// ---- GlobalTextList.TcGTLO
TEXTLIST GlobalTextList
  808 = '  +'
  159 = '  -'
  440 = ' +'
  1026 = ' -'
  1635 = '%0.2f'
  824 = '%i'
  778 = '+'
  2003 = '-'
  1760 = '1'
  225 = '2'
  751 = 'ACTUADORES'
  905 = 'Almacen'
  381 = 'Almacén'
  135 = 'Automático'
  67 = 'Azul'
  613 = 'Belt_Conveyor_2m_1'
  919 = 'Belt_conveyor_2m_1'
  114 = 'Belt_Conveyor_2m_2'
  119 = 'Belt_Conveyor_2m_3'
  170 = 'Belt_Conveyor_2m_4'
  987 = 'Belt_Conveyor_2m_5'
  96 = 'Belt_Conveyor_2m_6'
  269 = 'Belt_Conveyor_2m_7'
  285 = 'Belt_Conveyor_2m_8'
  759 = 'Belt_conveyor_4m_1'
  776 = 'Belt_Conveyor_4m_3'
  836 = 'Belt_Conveyor_4m_4'
  755 = 'Belt_Conveyor_4m_5'
  724 = 'Belt_Conveyor_4m_6'
  643 = 'Belt_conveyor_6m_1'
  497 = 'Belt_Conveyor_6m_2'
  202 = 'Belt_conveyor_6m_4'
  731 = 'Belt_conveyor_6m_5'
  768 = 'Belt_Conveyor_Inclined_1'
  535 = 'BL'
  1577 = 'Brazo'
  234 = 'Chain_Transfer_1_+'
  916 = 'Cinturon +'
  165 = 'Cinturón -'
  278 = 'Clamped base'
  1647 = 'Clamped der'
  321 = 'Clamped izq'
  82 = 'Clamped top'
  420 = 'Comienzo Linea Azul'
  1467 = 'Comienzo Produccion'
  78 = 'Comienzo Producción Azul'
  1309 = 'Command'
  1035 = 'Command ID'
  1959 = 'Control Almacen'
  1204 = 'Control Machines Centers'
  429 = 'Curved_Belt_Conveyor_1_CW'
  62 = 'Curved_Belt_Conveyor_2_CCW'
  578 = 'Curved_Roller_Conveyor_1_ccw'
  624 = 'Curved_Roller_Conveyor_2_ccw'
  222 = 'Descarte'
  1837 = 'Diffuse_Sensor_0'
  448 = 'Diffuse_Sensor_1'
  935 = 'Diffuse_Sensor_2'
  516 = 'Diffuse_Sensor_3'
  913 = 'Diffuse_Sensor_39'
  816 = 'Diffuse_Sensor_4'
  1082 = 'Diffuse_Sensor_41'
  895 = 'Diffuse_Sensor_43'
  528 = 'Diffuse_Sensor_44'
  482 = 'Diffuse_Sensor_5'
  68 = 'Diffuse_Sensor_8'
  560 = 'Emergency Stop'
  121 = 'Emergency Stop_1'
  284 = 'Emergency Stop_2'
  433 = 'Emisión'
  952 = 'Emisor'
  925 = 'Entrada'
  355 = 'Entrada Almacen'
  36 = 'Error RFID'
  683 = 'Extracción'
  1129 = 'f'
  120 = 'Final Linea Azul'
  1722 = 'Final Producción Azul'
  1140 = 'FL'
  296 = 'Flujo'
  363 = 'G'
  176 = 'gggg'
  131 = 'Giro Brazo'
  1627 = 'Giro Cinturon +'
  644 = 'Global'
  1976 = 'Grua'
  414 = 'hhhh'
  534 = 'inea Verde'
  546 = 'L'
  426 = 'Linea Almacen'
  588 = 'Linea Azul'
  456 = 'Linea Metal'
  439 = 'Linea Verde'
  1440 = 'Loading_Conveyor_1'
  1444 = 'Línea Almacén'
  386 = 'Machining_Center_1_Error'
  558 = 'Machining_Center_1_IsBusy'
  780 = 'Machining_Center_1_Opened'
  323 = 'Machining_Center_1_Produce_Lids'
  520 = 'Machining_Center_1_Progress'
  183 = 'Machining_Center_2_Error'
  615 = 'Machining_Center_2_IsBusy'
  617 = 'Machining_Center_2_Opened'
  1000 = 'Machining_Center_2_Produce_Lids'
  413 = 'Machining_Center_2_Progress'
  888 = 'Manual'
  1021 = 'Memory Index'
  1807 = 'ML'
  809 = 'Open_Door'
  105 = 'Open_Door_1'
  19 = 'Open_Door_2'
  976 = 'Palletizer'
  334 = 'Palletizer_1_Back_Limit'
  602 = 'Palletizer_1_Belt+'
  1173 = 'Palletizer_1_Belt-'
  536 = 'Palletizer_1_Chain+'
  942 = 'Palletizer_1_Chain-'
  1048 = 'Palletizer_1_Clamp'
  182 = 'Palletizer_1_Clamped'
  847 = 'Palletizer_1_Elevator+'
  108 = 'Palletizer_1_Elevator-'
  61 = 'Palletizer_1_Elevator_Moving'
  599 = 'Palletizer_1_Front_Limit'
  587 = 'Palletizer_1_MoveToLimit'
  124 = 'Palletizer_1_Open_Plate'
  557 = 'Palletizer_1_Plate_Limit'
  965 = 'Palletizer_1_Push'
  361 = 'Palletizer_1_Pusher_Limit'
  418 = 'Palletizer_1_Turn'
  404 = 'Pantalla Principal'
  897 = 'Pick & Place'
  1779 = 'Pinza'
  480 = 'Pivot_Arm_Sorter_1_Belt+'
  784 = 'Pivot_Arm_Sorter_1_Belt-'
  929 = 'Pivot_Arm_Sorter_1_Turn'
  302 = 'Pivot_Arm_Sorter_2_Belt+'
  744 = 'Pivot_Arm_Sorter_2_Belt-'
  614 = 'Pivot_Arm_Sorter_2_Turn'
  719 = 'Posición'
  762 = 'Principal'
  88 = 'Pusher_1'
  657 = 'Pusher_1_Back_Limit'
  45 = 'Pusher_1_Front_Limit'
  934 = 'Pusher_2'
  621 = 'Pusher_2_Back_Limit'
  774 = 'Pusher_2_Front_Limit'
  140 = 'Pusher_3'
  585 = 'Pusher_3_Back_Limit'
  306 = 'Pusher_3_Front_Limit'
  1770 = 'R'
  411 = 'Read Data'
  111 = 'Reset'
  1365 = 'Retroreflective_Sensor_1'
  331 = 'Retroreflective_Sensor_2'
  308 = 'RFID_Reader_1_Command'
  899 = 'RFID_Reader_1_Command_ID'
  459 = 'RFID_Reader_1_Ejecute_Command'
  1031 = 'RFID_Reader_1_Memory_Data'
  817 = 'RFID_Reader_1_Read_Data'
  377 = 'RFID_Reader_1_Status'
  874 = 'RFID_Reader_1_Writead_Data'
  508 = 'RFID_Reader_1_Write_Data'
  569 = 'Right_Positioner_1_Clamp'
  850 = 'Right_Positioner_1_Clamped'
  989 = 'Right_Positioner_1_Limit'
  523 = 'Right_Positioner_1_Raise'
  511 = 'Right_Positioner_2_Clamped'
  14 = 'Right_Positioner_2_Limit'
  620 = 'Roller_Conveyor_2m_1'
  251 = 'Roller_Conveyor_2m_2'
  1642 = 'Roller_Conveyor_2m_5'
  97 = 'Roller_Conveyor_2m_8'
  29 = 'Roller_Conveyor_4m_1'
  855 = 'Roller_Conveyor_4m_2'
  960 = 'Roller_Conveyor_4m_3'
  653 = 'Roller_Conveyor_6m_1'
  1263 = 'Roller_Conveyor_6m_2'
  627 = 'SENSORES'
  790 = 'Señales'
  1143 = 'Stacker_Crane_Left'
  1650 = 'Stacker_Crane_Left_Limit'
  1364 = 'Stacker_Crane_Lift'
  1622 = 'Stacker_Crane_Middle_Limit'
  1210 = 'Stacker_Crane_Moving_X'
  953 = 'Stacker_Crane_Moving_Z'
  1284 = 'Stacker_Crane_Right'
  380 = 'Stacker_Crane_Right_Limit'
  46 = 'Start'
  1155 = 'Start_1'
  1180 = 'Start_2'
  1706 = 'Status'
  769 = 'Stop'
  1228 = 'Stop_1'
  431 = 'Stop_2'
  518 = 'Turntable_1_Back_Limit'
  666 = 'Turntable_1_Front_Limit'
  556 = 'Turntable_1_Limit_0'
  77 = 'Turntable_1_Limit_90'
  1318 = 'Turntable_1_Roll_+'
  292 = 'Turntable_1_Roll_-'
  1288 = 'Turntable_1_Turn'
  1524 = 'Turntable_2_Back_Limit'
  1270 = 'Turntable_2_Front_Limit'
  235 = 'Turntable_2_Limit_0'
  473 = 'Turntable_2_Limit_90'
  1052 = 'Turntable_2_Roll_+'
  552 = 'Turntable_2_Roll_-'
  1580 = 'Turntable_2_Turn'
  337 = 'Two-Axis_Pick_Place_1_Detected'
  814 = 'Two-Axis_Pick_Place_1_Grab'
  112 = 'Two-Axis_Pick_Place_1_Gripper_CCW'
  309 = 'Two-Axis_Pick_Place_1_Gripper_CW'
  956 = 'Two-Axis_Pick_Place_1_Gripper_Rotating'
  811 = 'Two-Axis_Pick_Place_1_Moving_X'
  353 = 'Two-Axis_Pick_Place_1_Moving_Z'
  870 = 'Two-Axis_Pick_Place_1_Rotate'
  893 = 'Two-Axis_Pick_Place_1_Rotate_CCW'
  681 = 'Two-Axis_Pick_Place_1_Rotate_CW'
  541 = 'Two-Axis_Pick_Place_1_Rotating'
  568 = 'Two-Axis_Pick_Place_1_X'
  184 = 'Two-Axis_Pick_Place_1_Z'
  1262 = 'Two_Axis_Pick&Place'
  356 = 'Variables'
  810 = 'Vision_Sensor_1'
  288 = 'Vision_Sensor_10'
  21 = 'Vision_Sensor_11'
  936 = 'Vision_Sensor_12'
  53 = 'Vision_Sensor_13'
  669 = 'Vision_Sensor_14'
  985 = 'Vision_Sensor_15'
  999 = 'Vision_Sensor_4'
  357 = 'Vision_Sensor_40'
  996 = 'Vision_Sensor_42'
  84 = 'Vision_Sensor_5'
  841 = 'Vision_Sensor_6'
  335 = 'Vision_Sensor_7'
  688 = 'Vision_Sensor_8'
  43 = 'Vision_Sensor_9'
  1093 = 'vvvvvvvv'
  1646 = 'Write Data'
  1531 = 'Zona Inferior'
  909 = 'Zona Superior'
  805 = '¿Como introduzco valores?'
END_TEXTLIST

// ---- VISUs/Manual/Almacen_Manual.TcVIS
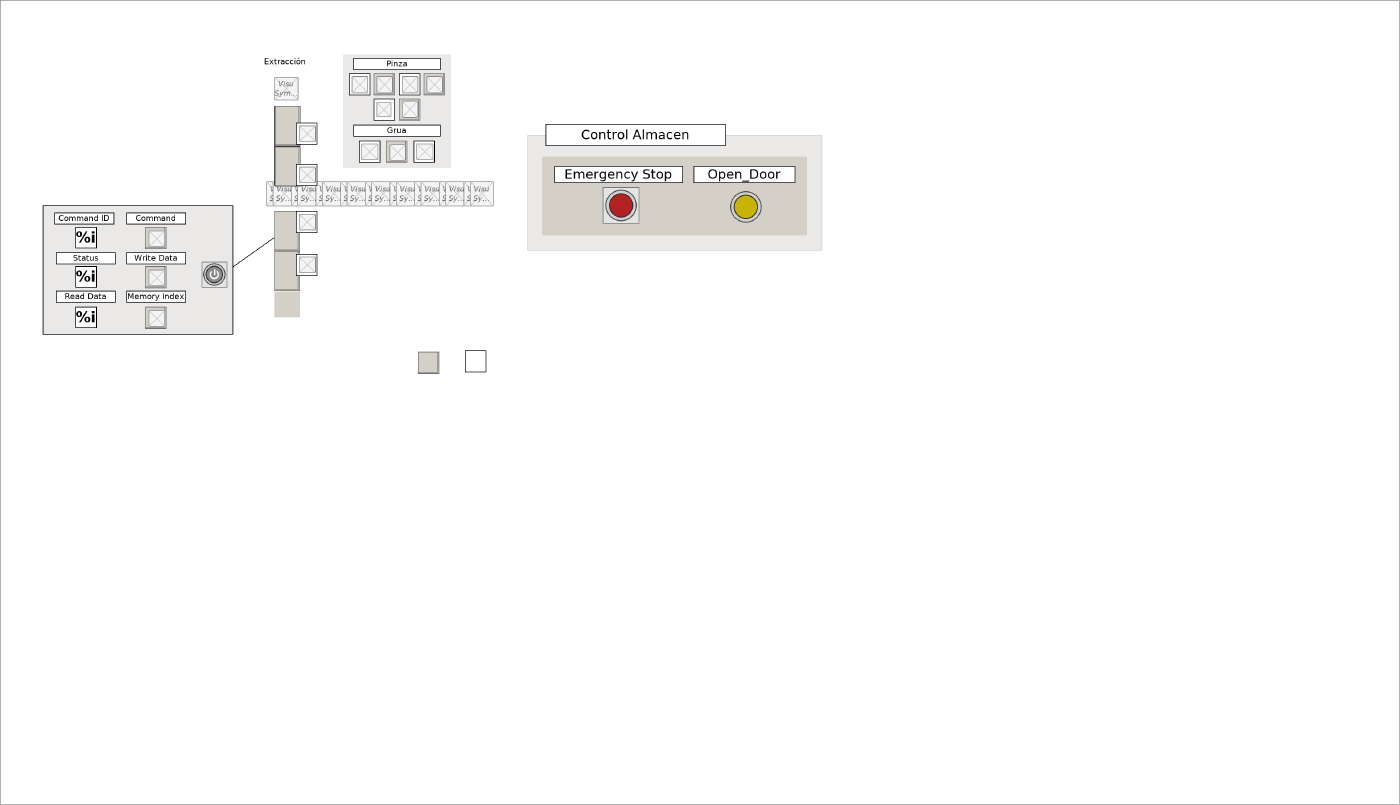
VISUALIZATION Almacen_Manual  // 1930x1110
    Rectangle (369,356 55x35), angle 90
    Group (367,250 330x48)
        Group (0,0 126x48)
            Group (0,0 92x48)
                Group (0,0 58x48)
                    Rectangle (8,5 24x23)
                    Image (0,0 32x34), image: VisuSymbols.Symbols.ArrowForward
                    Image (9,0 32x34), angle 90, image: VisuSymbols.Symbols.ArrowDown
                Group (34,0 58x48)
                    Rectangle (8,5 24x23)
                    Image (0,0 32x34), image: VisuSymbols.Symbols.ArrowForward
                    Image (9,0 32x34), angle 90, image: VisuSymbols.Symbols.ArrowDown
            Group (68,0 58x48)
                Rectangle (8,5 24x23)
                Image (0,0 32x34), image: VisuSymbols.Symbols.ArrowForward
                Image (9,0 32x34), angle 90, image: VisuSymbols.Symbols.ArrowDown
        Group (102,0 126x48)
            Group (0,0 92x48)
                Group (0,0 58x48)
                    Rectangle (8,5 24x23)
                    Image (0,0 32x34), image: VisuSymbols.Symbols.ArrowForward
                    Image (9,0 32x34), angle 90, image: VisuSymbols.Symbols.ArrowDown
                Group (34,0 58x48)
                    Rectangle (8,5 24x23)
                    Image (0,0 32x34), image: VisuSymbols.Symbols.ArrowForward
                    Image (9,0 32x34), angle 90, image: VisuSymbols.Symbols.ArrowDown
            Group (68,0 58x48)
                Rectangle (8,5 24x23)
                Image (0,0 32x34), image: VisuSymbols.Symbols.ArrowForward
                Image (9,0 32x34), angle 90, image: VisuSymbols.Symbols.ArrowDown
        Group (204,0 126x48)
            Group (0,0 92x48)
                Group (0,0 58x48)
                    Rectangle (8,5 24x23)
                    Image (0,0 32x34), image: VisuSymbols.Symbols.ArrowForward
                    Image (9,0 32x34), angle 90, image: VisuSymbols.Symbols.ArrowDown
                Group (34,0 58x48)
                    Rectangle (8,5 24x23)
                    Image (0,0 32x34), image: VisuSymbols.Symbols.ArrowForward
                    Image (9,0 32x34), angle 90, image: VisuSymbols.Symbols.ArrowDown
            Group (68,0 58x48)
                Rectangle (8,5 24x23)
                Image (0,0 32x34), image: VisuSymbols.Symbols.ArrowForward
                Image (9,0 32x34), angle 90, image: VisuSymbols.Symbols.ArrowDown
    InvisibleInput (355,103 77x35)
    Image (378,106 33x32), image: VisuSymbols.Symbols.ForwardStandard
    Rectangle (347,76 92x18), "Extracción"
    Rectangle (379,402 35x35), angle 90
    Rectangle (369,301 55x35), angle 90
    Rectangle (369,211 55x35), angle 90
    Rectangle (369,156 55x35), angle 90
    InvisibleInput (1163,198 18x136)
    Line (377,328) (318,370)
    InvisibleInput (262,497 18x41)
    Rectangle (1771,538 159x406), angle 90
    Rectangle (752,171 248x30), "Control Almacen"
    Rectangle (1780,528 108x365), angle 90
    PushSwitch (831,258 50x50), variable: GVL.Emergency_Stop_9, behaviour: TOGGLE, style: Switch-PushSwitch-Red
    Rectangle (764,229 177x23), "Emergency Stop"
    Lamp1 (1003,260 50x50), variable: NOT GVL.Safety_Door_13 OR NOT GVL.Safety_Door_14 OR NOT GVL.Safety_Door_15, style: Lamp-Lamp1-Yellow
    Rectangle (956,229 140x23), "Open_Door"
    Rectangle (1198,848 178x262), angle 90
    Rectangle (104,313 29x29), "%i", text variable: GVL.RFID_Reader_1_Command_ID
        p4168582468: GVL.RFID_Reader_1_Command_ID
    Rectangle (75,293 82x16), "Command ID"
    Rectangle (77,348 82x16), "Status"
    Rectangle (77,401 82x16), "Read Data"
    Rectangle (104,367 29x29), "%i", text variable: GVL.RFID_Reader_1_Status
        p4168582468: GVL.RFID_Reader_1_Status
    Rectangle (104,423 29x29), "%i", text variable: GVL.RFID_Reader_1_Read_Data
        p4168582468: GVL.RFID_Reader_1_Read_Data
    PowerSwitch (278,361 35x35), variable: GVL.RFID_Reader_1_Ejecute_Comm, behaviour: TOGGLE, style: Switch-PowerSwitch-Gray
    Button (378,346 35x55), colour toggle: GVL.Roller_Conveyor_2m_8, pressed state: GVL.Roller_Conveyor_2m_8
        OnMouseClick: toggle GVL.Roller_Conveyor_2m_8
    Button (378,291 35x55), colour toggle: GVL.Loading_Conveyor_1, pressed state: GVL.Loading_Conveyor_1
        OnMouseClick: toggle GVL.Loading_Conveyor_1
    Group (408,291 29x30), colour toggle: GVL.Retroreflective_Sensor_1
        RoundedRectangle (0,0 29x30), colour toggle: GVL.Diffuse_Sensor_4
        Image (4,4 23x22), image: VisuSymbols.Symbols.RSS1
    Group (408,350 29x30), colour toggle: GVL.Diffuse_Sensor_43
        RoundedRectangle (0,0 29x30), colour toggle: GVL.Diffuse_Sensor_4
        Image (4,4 23x22), image: VisuSymbols.Symbols.RSS1
    Button (379,202 35x55), colour toggle: GVL.Loading_Conveyor_2, pressed state: GVL.Loading_Conveyor_2
        OnMouseClick: toggle GVL.Loading_Conveyor_2
    Button (379,146 35x55), colour toggle: GVL.Roller_Conveyor_2m_9, pressed state: GVL.Roller_Conveyor_2m_9
        OnMouseClick: toggle GVL.Roller_Conveyor_2m_9
    Group (408,226 29x30), colour toggle: GVL.Retroreflective_Sensor_2
        RoundedRectangle (0,0 29x30), colour toggle: GVL.Diffuse_Sensor_4
        Image (4,4 23x22), image: VisuSymbols.Symbols.RSS1
    Group (408,169 29x30), colour toggle: GVL.Diffuse_Sensor_44
        RoundedRectangle (0,0 29x30), colour toggle: GVL.Diffuse_Sensor_4
        Image (4,4 23x22), image: VisuSymbols.Symbols.RSS1
    Rectangle (1505,647 156x148), angle 90
    Rectangle (487,80 120x16), "Pinza"
    Group (495,194 29x30), colour toggle: GVL.Stacker_Crane_1_Moving_X
        RoundedRectangle (0,0 29x30), colour toggle: GVL.Diffuse_Sensor_4
        Image (3,4 23x22), image: VisuSymbols.Symbols.DoubleArrow3
    Group (570,194 29x30), colour toggle: GVL.Stacker_Crane_1_Moving_Z
        RoundedRectangle (0,0 29x30), colour toggle: GVL.Diffuse_Sensor_4
        Image (4,4 23x22), image: VisuSymbols.Symbols.DoubleArrow4
    Rectangle (487,172 120x16), "Grua"
    Group (550,136 29x30), colour toggle: GVL.Stacker_Crane_1_Lift
        OnMouseClick: toggle GVL.Stacker_Crane_1_Lift
        Button (0,0 29x30), colour toggle: GVL.Stacker_Crane_1_Lift
        Image (4,3 22x23), image: VisuSymbols.Symbols.ArrowBoldUp
    Button (515,101 29x30)
    Image (519,105 22x23), colour toggle: GVL.Stacker_Crane_1_Left, image: VisuSymbols.Symbols.ArrowBoldLeft
        OnMouseClick: toggle GVL.Stacker_Crane_1_Left
    Group (481,101 29x30), colour toggle: GVL.Stacker_Crane_1_Left_Limit
        RoundedRectangle (0,0 29x30), colour toggle: GVL.Diffuse_Sensor_4
        Image (4,4 22x23), image: VisuSymbols.Symbols.ArrowBoldLeft
    Group (584,101 29x30), colour toggle: GVL.Stacker_Crane_1_Right
        OnMouseClick: toggle GVL.Stacker_Crane_1_Right
        Button (0,0 29x30)
        Image (4,4 22x23), image: VisuSymbols.Symbols.ArrowBoldRight
    Group (550,101 29x30), colour toggle: GVL.Stacker_Crane_1_Right_Limit
        RoundedRectangle (0,0 29x30), colour toggle: GVL.Diffuse_Sensor_4
        Image (4,4 22x23), image: VisuSymbols.Symbols.ArrowBoldRight
    Group (515,136 29x30), colour toggle: NOT GVL.Stacker_Crane_1_Middle_Limit
        RoundedRectangle (0,0 29x30), colour toggle: GVL.Diffuse_Sensor_4
        Image (4,5 20x20), angle 135, image: VisuSymbols.Symbols.DoubleArrow1
    Rectangle (174,293 82x16), "Command"
    Rectangle (174,348 82x16), "Write Data"
    Rectangle (174,401 82x16), "Memory Index"
    Group (200,313 29x30)
        OnMouseClick: write GVL.RFID_Reader_4_Command_ID via VisuDialogs.Numpad, min 0, max 100, format %i
        Button (0,0 29x30), text variable: GVL.RFID_Reader_1_Command
            OnMouseClick: write GVL.RFID_Reader_4_Command_ID via VisuDialogs.Numpad, min 0, max 100, format %i
        Image (5,5 22x22), image: VisuSymbols.Symbols.Edit
    Group (200,367 29x30)
        OnMouseClick: write GVL.RFID_Reader_4_Write_Data via VisuDialogs.Numpad, min 0, max 100, format %i
        Button (0,0 29x30), text variable: GVL.RFID_Reader_1_Command
            OnMouseClick: write GVL.RFID_Reader_4_Command_ID via VisuDialogs.Numpad, min 0, max 100, format %i
        Image (5,5 22x22), image: VisuSymbols.Symbols.Edit
    Group (200,423 29x30)
        OnMouseClick: write GVL.RFID_Reader_4_Memory_Index via VisuDialogs.Numpad, min 0, max 100, format %i
        Button (0,0 29x30), text variable: GVL.RFID_Reader_1_Command
            OnMouseClick: write GVL.RFID_Reader_4_Command_ID via VisuDialogs.Numpad, min 0, max 100, format %i
        Image (5,5 22x22), image: VisuSymbols.Symbols.Edit
    Group (532,194 29x30)
        OnMouseClick: write GVL.Stacker_Crane_1_Target_Position via VisuDialogs.Numpad, min 0, max 53, format %i
        Button (0,0 29x30), text variable: GVL.RFID_Reader_1_Command
            OnMouseClick: write GVL.RFID_Reader_4_Command_ID via VisuDialogs.Numpad, min 0, max 100, format %i
        Image (5,5 22x22), image: VisuSymbols.Symbols.Edit
    Button (576,485 29x30), text variable: GVL.RFID_Reader_1_Command
        OnMouseClick: write GVL.RFID_Reader_4_Command_ID via VisuDialogs.Numpad, min 0, max 100, format %i
    RoundedRectangle (641,483 29x30), colour toggle: GVL.Diffuse_Sensor_4
END_VISUALIZATION

// ---- VISUs/Manual/Linea_Almacen_Manual.TcVIS
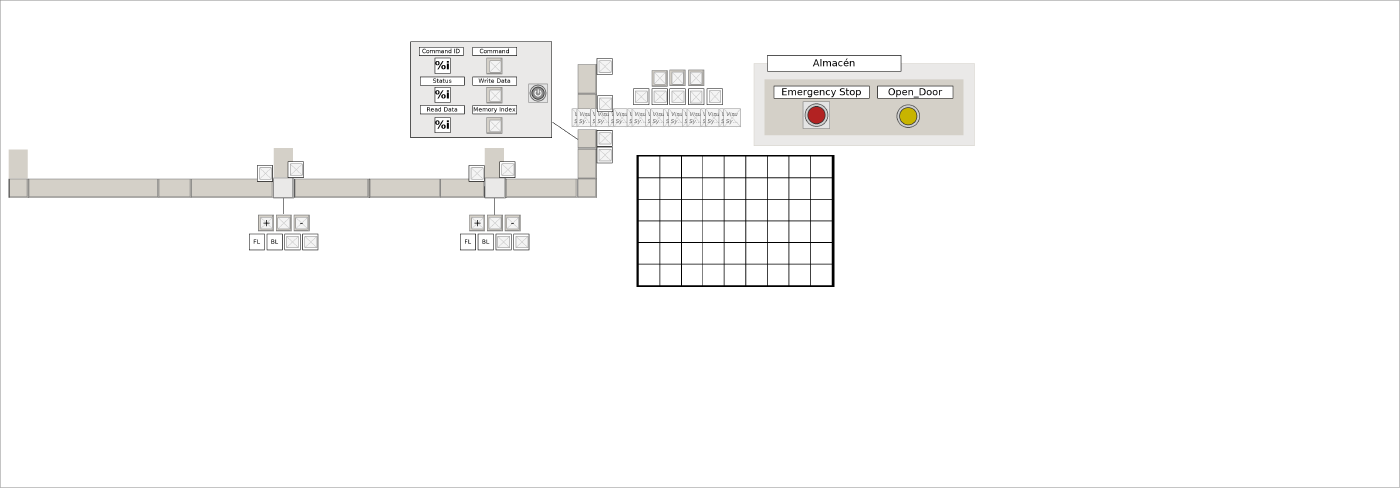
VISUALIZATION Linea_Almacen_Manual  // 2593x904
    Line (916,352) (916,399)
    Rectangle (889,284 55x35), angle 90
    Rectangle (155,228 35x241), angle 90
    Rectangle (984,282 35x132), angle 90
    Rectangle (306,318 35x60), angle 90
    Rectangle (412,272 35x152), angle 90
    Rectangle (506,329 38x38), angle 90
    Rectangle (597,280 35x137), angle 90
    Rectangle (732,283 35x131), angle 90
    Rectangle (839,308 35x81), angle 90
    Rectangle (906,336 21x38), angle 90
    Rectangle (17,331 35x35), angle 90
    Rectangle (8,286 53x35), angle 90
    Rectangle (498,284 54x35), angle 90
    Line (525,349) (525,396)
    InvisibleInput (1761,606 90x136)
    InvisibleInput (582,613 18x35)
    Button (17,331 35x35), colour toggle: GVL.Curved_Roller_Conveyor_1_CCW, pressed state: GVL.Curved_Roller_Conveyor_1_CCW
        OnMouseClick: toggle GVL.Curved_Roller_Conveyor_1_CCW
    Button (53,331 241x35), colour toggle: GVL.Roller_Conveyor_6m_1, pressed state: GVL.Roller_Conveyor_6m_1
        OnMouseClick: toggle GVL.Roller_Conveyor_6m_1
    Button (294,331 60x35), colour toggle: GVL.Chain_Transfer_1_mas, pressed state: GVL.Chain_Transfer_1_mas
        OnMouseClick: toggle GVL.Chain_Transfer_1_mas
    Button (354,331 152x35), colour toggle: GVL.Roller_Conveyor_4m_1, pressed state: GVL.Roller_Conveyor_4m_1
        OnMouseClick: toggle GVL.Roller_Conveyor_4m_1
    Button (506,329 38x38), pressed state: GVL.Roller_Conveyor_2m_2
    Button (546,331 137x35), colour toggle: GVL.Roller_Conveyor_6m_2, pressed state: GVL.Roller_Conveyor_6m_2
        OnMouseClick: toggle GVL.Roller_Conveyor_6m_2
    Button (685,331 131x35), colour toggle: GVL.Roller_Conveyor_4m_2, pressed state: GVL.Roller_Conveyor_4m_2
        OnMouseClick: toggle GVL.Roller_Conveyor_4m_2
    Button (816,331 81x35), colour toggle: GVL.Roller_Conveyor_2m_5, pressed state: GVL.Roller_Conveyor_2m_5
        OnMouseClick: toggle GVL.Roller_Conveyor_2m_5
    Button (898,329 38x38), colour toggle: GVL.Roller_Conveyor_2m_2, pressed state: GVL.Roller_Conveyor_2m_2
    Button (938,331 131x35), colour toggle: GVL.Roller_Conveyor_2m_2, pressed state: GVL.Roller_Conveyor_2m_2
        OnMouseClick: toggle GVL.Roller_Conveyor_2m_2
    Button (1070,331 35x35), colour toggle: GVL.Curved_Roller_Conveyor_2_CW, pressed state: GVL.Curved_Roller_Conveyor_2_CW
        OnMouseClick: toggle GVL.Curved_Roller_Conveyor_2_CW
    Button (1070,276 35x55), colour toggle: GVL.Roller_Conveyor_2m_8, pressed state: GVL.Roller_Conveyor_2m_8
        OnMouseClick: toggle GVL.Roller_Conveyor_2m_8
    Button (1070,240 35x35), colour toggle: GVL.Loading_Conveyor_1, pressed state: GVL.Loading_Conveyor_1
        OnMouseClick: toggle GVL.Loading_Conveyor_1
    Button (1070,174 35x35), colour toggle: GVL.Loading_Conveyor_2, pressed state: GVL.Loading_Conveyor_2
        OnMouseClick: toggle GVL.Loading_Conveyor_2
    Button (1070,119 35x55), colour toggle: GVL.Roller_Conveyor_2m_9, pressed state: GVL.Roller_Conveyor_2m_8
        OnMouseClick: toggle GVL.Roller_Conveyor_2m_9
    Rectangle (1179,287 366x244)
    Rectangle (1302,289 40x40)
    Rectangle (1302,329 40x40)
    Rectangle (1302,369 40x40)
    Rectangle (1302,409 40x40)
    Rectangle (1302,449 40x40)
    Rectangle (1302,489 40x40)
    Rectangle (1342,289 40x40)
    Rectangle (1342,329 40x40)
    Rectangle (1342,369 40x40)
    Rectangle (1342,409 40x40)
    Rectangle (1342,449 40x40)
    Rectangle (1342,489 40x40)
    Rectangle (1382,289 40x40)
    Rectangle (1382,329 40x40)
    Rectangle (1382,369 40x40)
    Rectangle (1382,409 40x40)
    Rectangle (1382,449 40x40)
    Rectangle (1382,489 40x40)
    Rectangle (1422,289 40x40)
    Rectangle (1422,329 40x40)
    Rectangle (1422,369 40x40)
    Rectangle (1422,409 40x40)
    Rectangle (1422,449 40x40)
    Rectangle (1422,489 40x40)
    Rectangle (1462,289 40x40)
    Rectangle (1462,329 40x40)
    Rectangle (1462,369 40x40)
    Rectangle (1462,409 40x40)
    Rectangle (1462,449 40x40)
    Rectangle (1462,489 40x40)
    Rectangle (1502,289 40x40)
    Rectangle (1502,329 40x40)
    Rectangle (1502,369 40x40)
    Rectangle (1502,409 40x40)
    Rectangle (1502,449 40x40)
    Rectangle (1502,489 40x40)
    Rectangle (1182,289 40x40)
    Rectangle (1182,329 40x40)
    Rectangle (1182,369 40x40)
    Rectangle (1182,409 40x40)
    Rectangle (1182,449 40x40)
    Rectangle (1182,489 40x40)
    Rectangle (1222,289 40x40)
    Rectangle (1222,329 40x40)
    Rectangle (1222,369 40x40)
    Rectangle (1222,409 40x40)
    Rectangle (1222,449 40x40)
    Rectangle (1222,489 40x40)
    Rectangle (1262,289 40x40)
    Rectangle (1262,329 40x40)
    Rectangle (1262,369 40x40)
    Rectangle (1262,409 40x40)
    Rectangle (1262,449 40x40)
    Rectangle (1262,489 40x40)
    Rectangle (1182,289 40x40), colour toggle: GVL.Clasificados[45].Visibilidad_Azul, invisible if: GVL.Clasificados[45].Visibilidad_Azul
    Rectangle (1182,329 40x40), colour toggle: GVL.Clasificados[36].Visibilidad_Azul, invisible if: GVL.Clasificados[36].Visibilidad_Azul
    Rectangle (1182,369 40x40), colour toggle: GVL.Clasificados[27].Visibilidad_Azul, invisible if: GVL.Clasificados[27].Visibilidad_Azul
    Rectangle (1182,409 40x40), colour toggle: GVL.Clasificados[18].Visibilidad_Azul, invisible if: GVL.Clasificados[18].Visibilidad_Azul
    Rectangle (1182,449 40x40), colour toggle: GVL.Clasificados[9].Visibilidad_Azul, invisible if: GVL.Clasificados[9].Visibilidad_Azul
    Rectangle (1182,489 40x40), colour toggle: GVL.Clasificados[0].Visibilidad_Azul, invisible if: GVL.Clasificados[0].Visibilidad_Azul
    Rectangle (1222,290 40x40)
    Rectangle (1222,330 40x40)
    Rectangle (1222,370 40x40)
    Rectangle (1222,410 40x40)
    Rectangle (1222,450 40x40)
    Rectangle (1222,490 40x40)
    Rectangle (1222,289 40x40), colour toggle: GVL.Clasificados[46].Visibilidad_Azul, invisible if: GVL.Clasificados[46].Visibilidad_Azul
    Rectangle (1222,329 40x40), colour toggle: GVL.Clasificados[37].Visibilidad_Azul, invisible if: GVL.Clasificados[37].Visibilidad_Azul
    Rectangle (1222,369 40x40), colour toggle: GVL.Clasificados[28].Visibilidad_Azul, invisible if: GVL.Clasificados[28].Visibilidad_Azul
    Rectangle (1222,409 40x40), colour toggle: GVL.Clasificados[19].Visibilidad_Azul, invisible if: GVL.Clasificados[19]Visibilidad_Azul
    Rectangle (1222,449 40x40), colour toggle: GVL.Clasificados[10].Visibilidad_Azul, invisible if: GVL.Clasificados[10].Visibilidad_Azul
    Rectangle (1222,489 40x40), colour toggle: GVL.Clasificados[1].Visibilidad_Azul, invisible if: GVL.Clasificados[1].Visibilidad_Azul
    Rectangle (1262,289 40x40)
    Rectangle (1262,329 40x40)
    Rectangle (1262,369 40x40)
    Rectangle (1262,409 40x40)
    Rectangle (1262,449 40x40)
    Rectangle (1262,489 40x40)
    Rectangle (1262,289 40x40), colour toggle: GVL.Clasificados[47].Visibilidad_Azul, invisible if: GVL.Clasificados[47].Visibilidad_Azul
    Rectangle (1262,329 40x40), colour toggle: GVL.Clasificados[38].Visibilidad_Azul, invisible if: GVL.Clasificados[38].Visibilidad_Azul
    Rectangle (1262,369 40x40), colour toggle: GVL.Clasificados[29].Visibilidad_Azul, invisible if: GVL.Clasificados[29].Visibilidad_Azul
    Rectangle (1262,409 40x40), colour toggle: GVL.Clasificados[20].Visibilidad_Azul, invisible if: GVL.Clasificados[20].Visibilidad_Azul
    Rectangle (1262,449 40x40), colour toggle: GVL.Clasificados[11].Visibilidad_Azul, invisible if: GVL.Clasificados[11].Visibilidad_Azul
    Rectangle (1262,489 40x40), colour toggle: GVL.Clasificados[2].Visibilidad_Azul, invisible if: GVL.Clasificados[2].Visibilidad_Azul
    Rectangle (1301,289 40x40)
    Rectangle (1301,329 40x40)
    Rectangle (1301,369 40x40)
    Rectangle (1301,409 40x40)
    Rectangle (1301,449 40x40)
    Rectangle (1301,489 40x40)
    Rectangle (1341,289 40x40)
    Rectangle (1341,329 40x40)
    Rectangle (1341,369 40x40)
    Rectangle (1341,409 40x40)
    Rectangle (1341,449 40x40)
    Rectangle (1341,489 40x40)
    Rectangle (1381,289 40x40)
    Rectangle (1381,329 40x40)
    Rectangle (1381,369 40x40)
    Rectangle (1381,409 40x40)
    Rectangle (1381,449 40x40)
    Rectangle (1381,489 40x40)
    Rectangle (1301,289 40x40), colour toggle: GVL.Clasificados[48].Visibilidad_Azul, invisible if: GVL.Clasificados[48].Visibilidad_Azul
    Rectangle (1301,329 40x40), colour toggle: GVL.Clasificados[39].Visibilidad_Azul, invisible if: GVL.Clasificados[39].Visibilidad_Azul
    Rectangle (1301,369 40x40), colour toggle: GVL.Clasificados[30].Visibilidad_Azul, invisible if: GVL.Clasificados[30].Visibilidad_Azul
    Rectangle (1301,409 40x40), colour toggle: GVL.Clasificados[21].Visibilidad_Azul, invisible if: GVL.Clasificados[21].Visibilidad_Azul
    Rectangle (1301,449 40x40), colour toggle: GVL.Clasificados[12].Visibilidad_Azul, invisible if: GVL.Clasificados[12].Visibilidad_Azul
    Rectangle (1301,489 40x40), colour toggle: GVL.Clasificados[3].Visibilidad_Azul, invisible if: GVL.Clasificados[3].Visibilidad_Azul
    Rectangle (1341,290 40x40)
    Rectangle (1341,330 40x40)
    Rectangle (1341,370 40x40)
    Rectangle (1341,410 40x40)
    Rectangle (1341,450 40x40)
    Rectangle (1341,490 40x40)
    Rectangle (1341,289 40x40), colour toggle: GVL.Clasificados[49].Visibilidad_Azul, invisible if: GVL.Clasificados[49].Visibilidad_Azul
    Rectangle (1341,329 40x40), colour toggle: GVL.Clasificados[40].Visibilidad_Azul, invisible if: GVL.Clasificados[40].Visibilidad_Azul
    Rectangle (1341,369 40x40), colour toggle: GVL.Clasificados[31].Visibilidad_Azul, invisible if: GVL.Clasificados[31].Visibilidad_Azul
    Rectangle (1341,409 40x40), colour toggle: GVL.Clasificados[22].Visibilidad_Azul, invisible if: GVL.Clasificados[22].Visibilidad_Azul
    Rectangle (1341,449 40x40), colour toggle: GVL.Clasificados[13].Visibilidad_Azul, invisible if: GVL.Clasificados[13].Visibilidad_Azul
    Rectangle (1341,489 40x40), colour toggle: GVL.Clasificados[4].Visibilidad_Azul, invisible if: GVL.Clasificados[4].Visibilidad_Azul
    Rectangle (1381,289 40x40)
    Rectangle (1381,329 40x40)
    Rectangle (1381,369 40x40)
    Rectangle (1381,409 40x40)
    Rectangle (1381,449 40x40)
    Rectangle (1381,489 40x40)
    Rectangle (1381,289 40x40), colour toggle: GVL.Clasificados[50].Visibilidad_Azul, invisible if: GVL.Clasificados[50].Visibilidad_Azul
    Rectangle (1381,329 40x40), colour toggle: GVL.Clasificados[41].Visibilidad_Azul, invisible if: GVL.Clasificados[41].Visibilidad_Azul
    Rectangle (1381,369 40x40), colour toggle: GVL.Clasificados[32].Visibilidad_Azul, invisible if: GVL.Clasificados[32].Visibilidad_Azul
    Rectangle (1381,409 40x40), colour toggle: GVL.Clasificados[23].Visibilidad_Azul, invisible if: GVL.Clasificados[23].Visibilidad_Azul
    Rectangle (1381,449 40x40), colour toggle: GVL.Clasificados[14].Visibilidad_Azul, invisible if: GVL.Clasificados[14].Visibilidad_Azul
    Rectangle (1381,489 40x40), colour toggle: GVL.Clasificados[5].Visibilidad_Azul, invisible if: GVL.Clasificados[5].Visibilidad_Azul
    Rectangle (1421,289 40x40)
    Rectangle (1421,329 40x40)
    Rectangle (1421,369 40x40)
    Rectangle (1421,409 40x40)
    Rectangle (1421,449 40x40)
    Rectangle (1421,489 40x40)
    Rectangle (1461,289 40x40)
    Rectangle (1461,329 40x40)
    Rectangle (1461,369 40x40)
    Rectangle (1461,409 40x40)
    Rectangle (1461,449 40x40)
    Rectangle (1461,489 40x40)
    Rectangle (1501,289 40x40)
    Rectangle (1501,329 40x40)
    Rectangle (1501,369 40x40)
    Rectangle (1501,409 40x40)
    Rectangle (1501,449 40x40)
    Rectangle (1501,489 40x40)
    Rectangle (1421,289 40x40), colour toggle: GVL.Clasificados[51].Visibilidad_Azul, invisible if: GVL.Clasificados[51].Visibilidad_Azul
    Rectangle (1421,329 40x40), colour toggle: GVL.Clasificados[42].Visibilidad_Azul, invisible if: GVL.Clasificados[42].Visibilidad_Azul
    Rectangle (1421,369 40x40), colour toggle: GVL.Clasificados[33].Visibilidad_Azul, invisible if: GVL.Clasificados[33].Visibilidad_Azul
    Rectangle (1421,409 40x40), colour toggle: GVL.Clasificados[24].Visibilidad_Azul, invisible if: GVL.Clasificados[24].Visibilidad_Azul
    Rectangle (1421,449 40x40), colour toggle: GVL.Clasificados[15].Visibilidad_Azul, invisible if: GVL.Clasificados[15].Visibilidad_Azul
    Rectangle (1421,489 40x40), colour toggle: GVL.Clasificados[6].Visibilidad_Azul, invisible if: GVL.Clasificados[6].Visibilidad_Azul
    Rectangle (1461,290 40x40)
    Rectangle (1461,330 40x40)
    Rectangle (1461,370 40x40)
    Rectangle (1461,410 40x40)
    Rectangle (1461,450 40x40)
    Rectangle (1461,490 40x40)
    Rectangle (1461,289 40x40), colour toggle: GVL.Clasificados[52].Visibilidad_Azul, invisible if: GVL.Clasificados[52].Visibilidad_Azul
    Rectangle (1461,329 40x40), colour toggle: GVL.Clasificados[43].Visibilidad_Azul, invisible if: GVL.Clasificados[43].Visibilidad_Azul
    Rectangle (1461,369 40x40), colour toggle: GVL.Clasificados[34].Visibilidad_Azul, invisible if: GVL.Clasificados[34].Visibilidad_Azul
    Rectangle (1461,409 40x40), colour toggle: GVL.Clasificados[25].Visibilidad_Azul, invisible if: GVL.Clasificados[25].Visibilidad_Azul
    Rectangle (1461,449 40x40), colour toggle: GVL.Clasificados[16].Visibilidad_Azul, invisible if: GVL.Clasificados[16].Visibilidad_Azul
    Rectangle (1461,489 40x40), colour toggle: GVL.Clasificados[7].Visibilidad_Azul, invisible if: GVL.Clasificados[7].Visibilidad_Azul
    Rectangle (1501,289 40x40)
    Rectangle (1501,329 40x40)
    Rectangle (1501,369 40x40)
    Rectangle (1501,409 40x40)
    Rectangle (1501,449 40x40)
    Rectangle (1501,489 40x40)
    Rectangle (1501,289 40x40), colour toggle: GVL.Clasificados[53].Visibilidad_Azul, invisible if: GVL.Clasificados[53].Visibilidad_Azul
    Rectangle (1501,329 40x40), colour toggle: GVL.Clasificados[44].Visibilidad_Azul, invisible if: GVL.Clasificados[44].Visibilidad_Azul
    Rectangle (1501,369 40x40), colour toggle: GVL.Clasificados[35].Visibilidad_Azul, invisible if: GVL.Clasificados[35].Visibilidad_Azul
    Rectangle (1501,409 40x40), colour toggle: GVL.Clasificados[26].Visibilidad_Azul, invisible if: GVL.Clasificados[26].Visibilidad_Azul
    Rectangle (1501,449 40x40), colour toggle: GVL.Clasificados[17].Visibilidad_Azul, invisible if: GVL.Clasificados[17].Visibilidad_Azul
    Rectangle (1501,489 40x40), colour toggle: GVL.Clasificados[8].Visibilidad_Azul, invisible if: GVL.Clasificados[8].Visibilidad_Azul
    Rectangle (1182,289 40x40), colour toggle: GVL.Clasificados[45].Visibilidad_Verde, invisible if: GVL.Clasificados[45].Visibilidad_Verde
    Rectangle (1182,329 40x40), colour toggle: GVL.Clasificados[36].Visibilidad_Verde, invisible if: GVL.Clasificados[36].Visibilidad_Verde
    Rectangle (1182,369 40x40), colour toggle: GVL.Clasificados[27].Visibilidad_Verde, invisible if: GVL.Clasificados[27].Visibilidad_Verde
    Rectangle (1182,409 40x40), colour toggle: GVL.Clasificados[18].Visibilidad_Verde, invisible if: GVL.Clasificados[18].Visibilidad_Verde
    Rectangle (1182,449 40x40), colour toggle: GVL.Clasificados[9].Visibilidad_Verde, invisible if: GVL.Clasificados[9].Visibilidad_Verde
    Rectangle (1182,489 40x40), colour toggle: GVL.Clasificados[0].Visibilidad_Verde, invisible if: GVL.Clasificados[0].Visibilidad_Verde
    Rectangle (1222,289 40x40), colour toggle: GVL.Clasificados[46].Visibilidad_Verde, invisible if: GVL.Clasificados[46].Visibilidad_Verde
    Rectangle (1222,329 40x40), colour toggle: GVL.Clasificados[37].Visibilidad_Verde, invisible if: GVL.Clasificados[37].Visibilidad_Verde
    Rectangle (1222,369 40x40), colour toggle: GVL.Clasificados[28].Visibilidad_Verde, invisible if: GVL.Clasificados[28].Visibilidad_Verde
    Rectangle (1222,409 40x40), colour toggle: GVL.Clasificados[19].Visibilidad_Verde, invisible if: GVL.Clasificados[19].Visibilidad_Verde
    Rectangle (1222,449 40x40), colour toggle: GVL.Clasificados[10].Visibilidad_Verde, invisible if: GVL.Clasificados[10].Visibilidad_Verde
    Rectangle (1222,489 40x40), colour toggle: GVL.Clasificados[1].Visibilidad_Verde, invisible if: GVL.Clasificados[1].Visibilidad_Verde
    Rectangle (1262,289 40x40), colour toggle: GVL.Clasificados[47].Visibilidad_Verde, invisible if: GVL.Clasificados[47].Visibilidad_Verde
    Rectangle (1262,329 40x40), colour toggle: GVL.Clasificados[38].Visibilidad_Verde, invisible if: GVL.Clasificados[38].Visibilidad_Verde
    Rectangle (1262,369 40x40), colour toggle: GVL.Clasificados[29].Visibilidad_Verde, invisible if: GVL.Clasificados[29].Visibilidad_Verde
    Rectangle (1262,409 40x40), colour toggle: GVL.Clasificados[20].Visibilidad_Verde, invisible if: GVL.Clasificados[20].Visibilidad_Verde
    Rectangle (1262,449 40x40), colour toggle: GVL.Clasificados[11].Visibilidad_Verde, invisible if: GVL.Clasificados[11].Visibilidad_Verde
    Rectangle (1262,489 40x40), colour toggle: GVL.Clasificados[2].Visibilidad_Verde, invisible if: GVL.Clasificados[2].Visibilidad_Verde
    Rectangle (1301,289 40x40), colour toggle: GVL.Clasificados[48].Visibilidad_Verde, invisible if: GVL.Clasificados[48].Visibilidad_Verde
    Rectangle (1301,329 40x40), colour toggle: GVL.Clasificados[39].Visibilidad_Verde, invisible if: GVL.Clasificados[39].Visibilidad_Verde
    Rectangle (1301,369 40x40), colour toggle: GVL.Clasificados[30].Visibilidad_Verde, invisible if: GVL.Clasificados[30].Visibilidad_Verde
    Rectangle (1301,409 40x40), colour toggle: GVL.Clasificados[21].Visibilidad_Verde, invisible if: GVL.Clasificados[21].Visibilidad_Verde
    Rectangle (1301,449 40x40), colour toggle: GVL.Clasificados[12].Visibilidad_Verde, invisible if: GVL.Clasificados[12].Visibilidad_Verde
    Rectangle (1301,489 40x40), colour toggle: GVL.Clasificados[3].Visibilidad_Verde, invisible if: GVL.Clasificados[3].Visibilidad_Verde
    Rectangle (1341,289 40x40), colour toggle: GVL.Clasificados[49].Visibilidad_Verde, invisible if: GVL.Clasificados[49].Visibilidad_Verde
    Rectangle (1341,329 40x40), colour toggle: GVL.Clasificados[40].Visibilidad_Verde, invisible if: GVL.Clasificados[40].Visibilidad_Verde
    Rectangle (1341,369 40x40), colour toggle: GVL.Clasificados[31].Visibilidad_Verde, invisible if: GVL.Clasificados[31].Visibilidad_Verde
    Rectangle (1341,409 40x40), colour toggle: GVL.Clasificados[22].Visibilidad_Verde, invisible if: GVL.Clasificados[22].Visibilidad_Verde
    Rectangle (1341,449 40x40), colour toggle: GVL.Clasificados[13].Visibilidad_Verde, invisible if: GVL.Clasificados[13].Visibilidad_Verde
    Rectangle (1341,489 40x40), colour toggle: GVL.Clasificados[4].Visibilidad_Verde, invisible if: GVL.Clasificados[4].Visibilidad_Verde
    Rectangle (1381,289 40x40), colour toggle: GVL.Clasificados[50].Visibilidad_Verde, invisible if: GVL.Clasificados[50].Visibilidad_Verde
    Rectangle (1381,329 40x40), colour toggle: GVL.Clasificados[41].Visibilidad_Verde, invisible if: GVL.Clasificados[41].Visibilidad_Verde
    Rectangle (1381,369 40x40), colour toggle: GVL.Clasificados[32].Visibilidad_Verde, invisible if: GVL.Clasificados[32].Visibilidad_Verde
    Rectangle (1381,409 40x40), colour toggle: GVL.Clasificados[23].Visibilidad_Verde, invisible if: GVL.Clasificados[23].Visibilidad_Verde
    Rectangle (1381,449 40x40), colour toggle: GVL.Clasificados[14].Visibilidad_Verde, invisible if: GVL.Clasificados[14].Visibilidad_Verde
    Rectangle (1381,489 40x40), colour toggle: GVL.Clasificados[5].Visibilidad_Verde, invisible if: GVL.Clasificados[5].Visibilidad_Verde
    Rectangle (1421,289 40x40), colour toggle: GVL.Clasificados[51].Visibilidad_Verde, invisible if: GVL.Clasificados[51].Visibilidad_Verde
    Rectangle (1421,329 40x40), colour toggle: GVL.Clasificados[42].Visibilidad_Verde, invisible if: GVL.Clasificados[42].Visibilidad_Verde
    Rectangle (1421,369 40x40), colour toggle: GVL.Clasificados[33].Visibilidad_Verde, invisible if: GVL.Clasificados[33].Visibilidad_Verde
    Rectangle (1421,409 40x40), colour toggle: GVL.Clasificados[24].Visibilidad_Verde, invisible if: GVL.Clasificados[24].Visibilidad_Verde
    Rectangle (1421,449 40x40), colour toggle: GVL.Clasificados[15].Visibilidad_Verde, invisible if: GVL.Clasificados[15].Visibilidad_Verde
    Rectangle (1421,489 40x40), colour toggle: GVL.Clasificados[6].Visibilidad_Verde, invisible if: GVL.Clasificados[6].Visibilidad_Verde
    Rectangle (1461,289 40x40), colour toggle: GVL.Clasificados[52].Visibilidad_Verde, invisible if: GVL.Clasificados[52].Visibilidad_Verde
    Rectangle (1461,329 40x40), colour toggle: GVL.Clasificados[43].Visibilidad_Verde, invisible if: GVL.Clasificados[43].Visibilidad_Verde
    Rectangle (1461,369 40x40), colour toggle: GVL.Clasificados[34].Visibilidad_Verde, invisible if: GVL.Clasificados[34].Visibilidad_Verde
    Rectangle (1461,409 40x40), colour toggle: GVL.Clasificados[25].Visibilidad_Verde, invisible if: GVL.Clasificados[25].Visibilidad_Verde
    Rectangle (1461,449 40x40), colour toggle: GVL.Clasificados[16].Visibilidad_Verde, invisible if: GVL.Clasificados[16].Visibilidad_Verde
    Rectangle (1461,489 40x40), colour toggle: GVL.Clasificados[7].Visibilidad_Verde, invisible if: GVL.Clasificados[7].Visibilidad_Verde
    Rectangle (1501,289 40x40), colour toggle: GVL.Clasificados[53].Visibilidad_Verde, invisible if: GVL.Clasificados[53].Visibilidad_Verde
    Rectangle (1501,329 40x40), colour toggle: GVL.Clasificados[44].Visibilidad_Verde, invisible if: GVL.Clasificados[44].Visibilidad_Verde
    Rectangle (1501,369 40x40), colour toggle: GVL.Clasificados[35].Visibilidad_Verde, invisible if: GVL.Clasificados[35].Visibilidad_Verde
    Rectangle (1501,409 40x40), colour toggle: GVL.Clasificados[26].Visibilidad_Verde, invisible if: GVL.Clasificados[26].Visibilidad_Verde
    Rectangle (1501,449 40x40), colour toggle: GVL.Clasificados[17].Visibilidad_Verde, invisible if: GVL.Clasificados[17].Visibilidad_Verde
    Rectangle (1501,489 40x40), colour toggle: GVL.Clasificados[8].Visibilidad_Verde, invisible if: GVL.Clasificados[8].Visibilidad_Verde
    Rectangle (1421,289 40x40), colour toggle: GVL.Clasificados[51].Visibilidad_Metal, invisible if: GVL.Clasificados[51].Visibilidad_Metal
    Rectangle (1421,369 40x40), colour toggle: GVL.Clasificados[33].Visibilidad_Metal, invisible if: GVL.Clasificados[33].Visibilidad_Metal
    Rectangle (1421,329 40x40), colour toggle: GVL.Clasificados[42].Visibilidad_Metal, invisible if: GVL.Clasificados[42].Visibilidad_Metal
    Rectangle (1421,409 40x40), colour toggle: GVL.Clasificados[24].Visibilidad_Metal, invisible if: GVL.Clasificados[24].Visibilidad_Metal
    Rectangle (1421,449 40x40), colour toggle: GVL.Clasificados[15].Visibilidad_Metal, invisible if: GVL.Clasificados[15].Visibilidad_Metal
    Rectangle (1421,489 40x40), colour toggle: GVL.Clasificados[6].Visibilidad_Metal, invisible if: GVL.Clasificados[6].Visibilidad_Metal
    Rectangle (1461,289 40x40), colour toggle: GVL.Clasificados[52].Visibilidad_Metal, invisible if: GVL.Clasificados[52].Visibilidad_Metal
    Rectangle (1461,369 40x40), colour toggle: GVL.Clasificados[34].Visibilidad_Metal, invisible if: GVL.Clasificados[34].Visibilidad_Metal
    Rectangle (1461,329 40x40), colour toggle: GVL.Clasificados[43].Visibilidad_Metal, invisible if: GVL.Clasificados[43].Visibilidad_Metal
    Rectangle (1461,409 40x40), colour toggle: GVL.Clasificados[25].Visibilidad_Metal, invisible if: GVL.Clasificados[25].Visibilidad_Metal
    Rectangle (1461,449 40x40), colour toggle: GVL.Clasificados[16].Visibilidad_Metal, invisible if: GVL.Clasificados[16].Visibilidad_Metal
    Rectangle (1461,489 40x40), colour toggle: GVL.Clasificados[7].Visibilidad_Metal, invisible if: GVL.Clasificados[7].Visibilidad_Metal
    Rectangle (1501,289 40x40), colour toggle: GVL.Clasificados[53].Visibilidad_Metal, invisible if: GVL.Clasificados[53].Visibilidad_Metal
    Rectangle (1501,369 40x40), colour toggle: GVL.Clasificados[35].Visibilidad_Metal, invisible if: GVL.Clasificados[35].Visibilidad_Metal
    Rectangle (1501,329 40x40), colour toggle: GVL.Clasificados[44].Visibilidad_Metal, invisible if: GVL.Clasificados[44].Visibilidad_Metal
    Rectangle (1501,409 40x40), colour toggle: GVL.Clasificados[26].Visibilidad_Metal, invisible if: GVL.Clasificados[26].Visibilidad_Metal
    Rectangle (1501,449 40x40), colour toggle: GVL.Clasificados[17].Visibilidad_Metal, invisible if: GVL.Clasificados[17].Visibilidad_Metal
    Rectangle (1501,489 40x40), colour toggle: GVL.Clasificados[8].Visibilidad_Metal, invisible if: GVL.Clasificados[8].Visibilidad_Metal
    Rectangle (1182,289 40x40), colour toggle: GVL.Clasificados[45].Visibilidad_Metal, invisible if: GVL.Clasificados[45].Visibilidad_Metal
    Rectangle (1182,369 40x40), colour toggle: GVL.Clasificados[27].Visibilidad_Metal, invisible if: GVL.Clasificados[27].Visibilidad_Metal
    Rectangle (1182,329 40x40), colour toggle: GVL.Clasificados[36].Visibilidad_Metal, invisible if: GVL.Clasificados[36].Visibilidad_Metal
    Rectangle (1182,409 40x40), colour toggle: GVL.Clasificados[18].Visibilidad_Metal, invisible if: GVL.Clasificados[18].Visibilidad_Metal
    Rectangle (1182,449 40x40), colour toggle: GVL.Clasificados[9].Visibilidad_Metal, invisible if: GVL.Clasificados[9].Visibilidad_Metal
    Rectangle (1182,489 40x40), colour toggle: GVL.Clasificados[0].Visibilidad_Metal, invisible if: GVL.Clasificados[0].Visibilidad_Metal
    Rectangle (1222,289 40x40), colour toggle: GVL.Clasificados[46].Visibilidad_Metal, invisible if: GVL.Clasificados[46].Visibilidad_Metal
    Rectangle (1222,369 40x40), colour toggle: GVL.Clasificados[28].Visibilidad_Metal, invisible if: GVL.Clasificados[28].Visibilidad_Metal
    Rectangle (1222,329 40x40), colour toggle: GVL.Clasificados[37].Visibilidad_Metal, invisible if: GVL.Clasificados[37].Visibilidad_Metal
    Rectangle (1222,409 40x40), colour toggle: GVL.Clasificados[19].Visibilidad_Metal, invisible if: GVL.Clasificados[19].Visibilidad_Metal
    Rectangle (1222,449 40x40), colour toggle: GVL.Clasificados[10].Visibilidad_Metal, invisible if: GVL.Clasificados[10].Visibilidad_Metal
    Rectangle (1222,489 40x40), colour toggle: GVL.Clasificados[1].Visibilidad_Metal, invisible if: GVL.Clasificados[1].Visibilidad_Metal
    Rectangle (1262,289 40x40), colour toggle: GVL.Clasificados[47].Visibilidad_Metal, invisible if: GVL.Clasificados[47].Visibilidad_Metal
    Rectangle (1262,369 40x40), colour toggle: GVL.Clasificados[29].Visibilidad_Metal, invisible if: GVL.Clasificados[29].Visibilidad_Metal
    Rectangle (1262,329 40x40), colour toggle: GVL.Clasificados[38].Visibilidad_Metal, invisible if: GVL.Clasificados[38].Visibilidad_Metal
    Rectangle (1262,409 40x40), colour toggle: GVL.Clasificados[20].Visibilidad_Metal, invisible if: GVL.Clasificados[20].Visibilidad_Metal
    Rectangle (1262,449 40x40), colour toggle: GVL.Clasificados[11].Visibilidad_Metal, invisible if: GVL.Clasificados[11].Visibilidad_Metal
    Rectangle (1262,489 40x40), colour toggle: GVL.Clasificados[2].Visibilidad_Metal, invisible if: GVL.Clasificados[2].Visibilidad_Metal
    Rectangle (1302,289 40x40), colour toggle: GVL.Clasificados[48].Visibilidad_Metal, invisible if: GVL.Clasificados[48].Visibilidad_Metal
    Rectangle (1302,369 40x40), colour toggle: GVL.Clasificados[30].Visibilidad_Metal, invisible if: GVL.Clasificados[30].Visibilidad_Metal
    Rectangle (1302,329 40x40), colour toggle: GVL.Clasificados[39].Visibilidad_Metal, invisible if: GVL.Clasificados[39].Visibilidad_Metal
    Rectangle (1302,409 40x40), colour toggle: GVL.Clasificados[21].Visibilidad_Metal, invisible if: GVL.Clasificados[21].Visibilidad_Metal
    Rectangle (1302,449 40x40), colour toggle: GVL.Clasificados[12].Visibilidad_Metal, invisible if: GVL.Clasificados[12].Visibilidad_Metal
    Rectangle (1302,489 40x40), colour toggle: GVL.Clasificados[3].Visibilidad_Metal, invisible if: GVL.Clasificados[3].Visibilidad_Metal
    Rectangle (1341,289 40x40), colour toggle: GVL.Clasificados[49].Visibilidad_Metal, invisible if: GVL.Clasificados[49 ].Visibilidad_Metal
    Rectangle (1341,369 40x40), colour toggle: GVL.Clasificados[31].Visibilidad_Metal, invisible if: GVL.Clasificados[31].Visibilidad_Metal
    Rectangle (1341,329 40x40), colour toggle: GVL.Clasificados[40].Visibilidad_Metal, invisible if: GVL.Clasificados[40].Visibilidad_Metal
    Rectangle (1341,409 40x40), colour toggle: GVL.Clasificados[22].Visibilidad_Metal, invisible if: GVL.Clasificados[22].Visibilidad_Metal
    Rectangle (1341,449 40x40), colour toggle: GVL.Clasificados[13].Visibilidad_Metal, invisible if: GVL.Clasificados[13].Visibilidad_Metal
    Rectangle (1341,489 40x40), colour toggle: GVL.Clasificados[4].Visibilidad_Metal, invisible if: GVL.Clasificados[4].Visibilidad_Metal
    Rectangle (1381,289 40x40), colour toggle: GVL.Clasificados[50].Visibilidad_Metal, invisible if: GVL.Clasificados[50].Visibilidad_Metal
    Rectangle (1381,369 40x40), colour toggle: GVL.Clasificados[32].Visibilidad_Metal, invisible if: GVL.Clasificados[32].Visibilidad_Metal
    Rectangle (1381,329 40x40), colour toggle: GVL.Clasificados[41].Visibilidad_Metal, invisible if: GVL.Clasificados[41].Visibilidad_Metal
    Rectangle (1381,409 40x40), colour toggle: GVL.Clasificados[23].Visibilidad_Metal, invisible if: GVL.Clasificados[23].Visibilidad_Metal
    Rectangle (1381,449 40x40), colour toggle: GVL.Clasificados[14].Visibilidad_Metal, invisible if: GVL.Clasificados[14].Visibilidad_Metal
    Rectangle (1381,489 40x40), colour toggle: GVL.Clasificados[5].Visibilidad_Metal, invisible if: GVL.Clasificados[5].Visibilidad_Metal
    Rectangle (1182,289 40x40), invisible if: GVL.Clasificados[45].Visibilidad_Vacio
    Rectangle (1182,329 40x40), invisible if: GVL.Clasificados[36].Visibilidad_Vacio
    Rectangle (1182,369 40x40), invisible if: GVL.Clasificados[27].Visibilidad_Vacio
    Rectangle (1182,409 40x40), invisible if: GVL.Clasificados[18].Visibilidad_Vacio
    Rectangle (1182,449 40x40), invisible if: GVL.Clasificados[9].Visibilidad_Vacio
    Rectangle (1182,489 40x40), invisible if: GVL.Clasificados[0].Visibilidad_Vacio
    Rectangle (1222,289 40x40), invisible if: GVL.Clasificados[46].Visibilidad_Vacio
    Rectangle (1222,329 40x40), invisible if: GVL.Clasificados[37].Visibilidad_Vacio
    Rectangle (1222,369 40x40), invisible if: GVL.Clasificados[28].Visibilidad_Vacio
    Rectangle (1222,409 40x40), invisible if: GVL.Clasificados[19].Visibilidad_Vacio
    Rectangle (1222,449 40x40), invisible if: GVL.Clasificados[10].Visibilidad_Vacio
    Rectangle (1222,489 40x40), invisible if: GVL.Clasificados[1].Visibilidad_Vacio
    Rectangle (1262,289 40x40), invisible if: GVL.Clasificados[47].Visibilidad_Vacio
    Rectangle (1262,329 40x40), invisible if: GVL.Clasificados[38].Visibilidad_Vacio
    Rectangle (1262,369 40x40), invisible if: GVL.Clasificados[29].Visibilidad_Vacio
    Rectangle (1262,409 40x40), invisible if: GVL.Clasificados[20].Visibilidad_Vacio
    Rectangle (1262,449 40x40), invisible if: GVL.Clasificados[11].Visibilidad_Vacio
    Rectangle (1262,489 40x40), invisible if: GVL.Clasificados[2].Visibilidad_Vacio
    Rectangle (1301,289 40x40), invisible if: GVL.Clasificados[48].Visibilidad_Vacio
    Rectangle (1301,329 40x40), invisible if: GVL.Clasificados[39].Visibilidad_Vacio
    Rectangle (1301,369 40x40), invisible if: GVL.Clasificados[30].Visibilidad_Vacio
    Rectangle (1301,409 40x40), invisible if: GVL.Clasificados[21].Visibilidad_Vacio
    Rectangle (1301,449 40x40), invisible if: GVL.Clasificados[12].Visibilidad_Vacio
    Rectangle (1301,489 40x40), invisible if: GVL.Clasificados[3].Visibilidad_Vacio
    Rectangle (1341,289 40x40), invisible if: GVL.Clasificados[49].Visibilidad_Vacio
    Rectangle (1341,329 40x40), invisible if: GVL.Clasificados[40].Visibilidad_Vacio
    Rectangle (1341,369 40x40), invisible if: GVL.Clasificados[31].Visibilidad_Vacio
    Rectangle (1341,409 40x40), invisible if: GVL.Clasificados[22].Visibilidad_Vacio
    Rectangle (1341,449 40x40), invisible if: GVL.Clasificados[13].Visibilidad_Vacio
    Rectangle (1341,489 40x40), invisible if: GVL.Clasificados[4].Visibilidad_Vacio
    Rectangle (1381,289 40x40), invisible if: GVL.Clasificados[50].Visibilidad_Vacio
    Rectangle (1381,329 40x40), invisible if: GVL.Clasificados[41].Visibilidad_Vacio
    Rectangle (1381,369 40x40), invisible if: GVL.Clasificados[32].Visibilidad_Vacio
    Rectangle (1381,409 40x40), invisible if: GVL.Clasificados[23].Visibilidad_Vacio
    Rectangle (1381,449 40x40), invisible if: GVL.Clasificados[14].Visibilidad_Vacio
    Rectangle (1381,489 40x40), invisible if: GVL.Clasificados[5].Visibilidad_Vacio
    Rectangle (1421,289 40x40), invisible if: GVL.Clasificados[51].Visibilidad_Vacio
    Rectangle (1421,329 40x40), invisible if: GVL.Clasificados[42].Visibilidad_Vacio
    Rectangle (1421,369 40x40), invisible if: GVL.Clasificados[33].Visibilidad_Vacio
    Rectangle (1421,409 40x40), invisible if: GVL.Clasificados[24].Visibilidad_Vacio
    Rectangle (1421,449 40x40), invisible if: GVL.Clasificados[15].Visibilidad_Vacio
    Rectangle (1421,489 40x40), invisible if: GVL.Clasificados[6].Visibilidad_Vacio
    Rectangle (1461,289 40x40), invisible if: GVL.Clasificados[52].Visibilidad_Vacio
    Rectangle (1461,329 40x40), invisible if: GVL.Clasificados[43].Visibilidad_Vacio
    Rectangle (1461,369 40x40), invisible if: GVL.Clasificados[34].Visibilidad_Vacio
    Rectangle (1461,409 40x40), invisible if: GVL.Clasificados[25].Visibilidad_Vacio
    Rectangle (1461,449 40x40), invisible if: GVL.Clasificados[16].Visibilidad_Vacio
    Rectangle (1461,489 40x40), invisible if: GVL.Clasificados[7].Visibilidad_Vacio
    Rectangle (1501,289 40x40), invisible if: GVL.Clasificados[53].Visibilidad_Vacio
    Rectangle (1501,329 40x40), invisible if: GVL.Clasificados[44].Visibilidad_Vacio
    Rectangle (1501,369 40x40), invisible if: GVL.Clasificados[35].Visibilidad_Vacio
    Rectangle (1501,409 40x40), invisible if: GVL.Clasificados[26].Visibilidad_Vacio
    Rectangle (1501,449 40x40), invisible if: GVL.Clasificados[17].Visibilidad_Vacio
    Rectangle (1501,489 40x40), invisible if: GVL.Clasificados[8].Visibilidad_Vacio
    Group (1059,201 330x48)
        Group (0,0 126x48)
            Group (0,0 92x48)
                Group (0,0 58x48)
                    Rectangle (8,5 24x23)
                    Image (0,0 32x34), image: VisuSymbols.Symbols.ArrowForward
                    Image (9,0 32x34), angle 90, image: VisuSymbols.Symbols.ArrowDown
                Group (34,0 58x48)
                    Rectangle (8,5 24x23)
                    Image (0,0 32x34), image: VisuSymbols.Symbols.ArrowForward
                    Image (9,0 32x34), angle 90, image: VisuSymbols.Symbols.ArrowDown
            Group (68,0 58x48)
                Rectangle (8,5 24x23)
                Image (0,0 32x34), image: VisuSymbols.Symbols.ArrowForward
                Image (9,0 32x34), angle 90, image: VisuSymbols.Symbols.ArrowDown
        Group (102,0 126x48)
            Group (0,0 92x48)
                Group (0,0 58x48)
                    Rectangle (8,5 24x23)
                    Image (0,0 32x34), image: VisuSymbols.Symbols.ArrowForward
                    Image (9,0 32x34), angle 90, image: VisuSymbols.Symbols.ArrowDown
                Group (34,0 58x48)
                    Rectangle (8,5 24x23)
                    Image (0,0 32x34), image: VisuSymbols.Symbols.ArrowForward
                    Image (9,0 32x34), angle 90, image: VisuSymbols.Symbols.ArrowDown
            Group (68,0 58x48)
                Rectangle (8,5 24x23)
                Image (0,0 32x34), image: VisuSymbols.Symbols.ArrowForward
                Image (9,0 32x34), angle 90, image: VisuSymbols.Symbols.ArrowDown
        Group (204,0 126x48)
            Group (0,0 92x48)
                Group (0,0 58x48)
                    Rectangle (8,5 24x23)
                    Image (0,0 32x34), image: VisuSymbols.Symbols.ArrowForward
                    Image (9,0 32x34), angle 90, image: VisuSymbols.Symbols.ArrowDown
                Group (34,0 58x48)
                    Rectangle (8,5 24x23)
                    Image (0,0 32x34), image: VisuSymbols.Symbols.ArrowForward
                    Image (9,0 32x34), angle 90, image: VisuSymbols.Symbols.ArrowDown
            Group (68,0 58x48)
                Rectangle (8,5 24x23)
                Image (0,0 32x34), image: VisuSymbols.Symbols.ArrowForward
                Image (9,0 32x34), angle 90, image: VisuSymbols.Symbols.ArrowDown
    Group (476,306 29x30), colour toggle: GVL.Diffuse_Sensor_39
        RoundedRectangle (0,0 29x30), colour toggle: GVL.Diffuse_Sensor_4
        Image (4,4 23x22), image: VisuSymbols.Symbols.RSS1
    Group (533,299 29x30), colour toggle: GVL.Diffuse_Sensor_40
        RoundedRectangle (0,0 29x30), colour toggle: GVL.Diffuse_Sensor_4
        Image (4,4 23x22), image: VisuSymbols.Symbols.RSS1
    Group (868,306 29x30), colour toggle: GVL.Diffuse_Sensor_41
        RoundedRectangle (0,0 29x30), colour toggle: GVL.Diffuse_Sensor_4
        Image (4,4 23x22), image: VisuSymbols.Symbols.RSS1
    Group (925,299 29x30), colour toggle: GVL.Diffuse_Sensor_42
        RoundedRectangle (0,0 29x30), colour toggle: GVL.Diffuse_Sensor_4
        Image (4,4 23x22), image: VisuSymbols.Symbols.RSS1
    Group (1106,177 29x30), colour toggle: GVL.Retroreflective_Sensor_2
        RoundedRectangle (0,0 29x30), colour toggle: GVL.Diffuse_Sensor_4
        Image (4,4 23x22), image: VisuSymbols.Symbols.RSS1
    Group (1105,108 29x30), colour toggle: GVL.Diffuse_Sensor_44
        RoundedRectangle (0,0 29x30), colour toggle: GVL.Diffuse_Sensor_4
        Image (4,4 23x22), image: VisuSymbols.Symbols.RSS1
    Group (1105,241 29x30), colour toggle: GVL.Retroreflective_Sensor_1
        RoundedRectangle (0,0 29x30), colour toggle: GVL.Diffuse_Sensor_4
        Image (4,4 23x22), image: VisuSymbols.Symbols.RSS1
    Group (1105,272 29x30), colour toggle: GVL.Diffuse_Sensor_43
        RoundedRectangle (0,0 29x30), colour toggle: GVL.Diffuse_Sensor_4
        Image (4,4 23x22), image: VisuSymbols.Symbols.RSS1
    Button (478,398 29x30), colour toggle: GVL.Turnable_1_Roll_mas, pressed state: GVL.Turnable_1_Roll_mas
        OnMouseClick: toggle GVL.Turnable_1_Roll_mas
    Image (482,402 23x22), "+", colour toggle: GVL.Turnable_1_Roll_mas, image: VisuSymbols.Symbols.ArrowRoundRightRight
        OnMouseClick: toggle GVL.Turnable_1_Roll_mas
    RoundedRectangle (461,433 29x30), "FL", colour toggle: GVL.Turnable_1_Front_Limit
    Button (511,398 29x30), colour toggle: GVL.Turnable_1_Turn, pressed state: GVL.Turnable_1_Turn
        OnMouseClick: toggle GVL.Turnable_1_Turn
    Image (514,402 23x22), colour toggle: GVL.Turnable_1_Turn, image: VisuSymbols.Symbols.ArrowCircle2LeftUpDown
        OnMouseClick: toggle GVL.Turnable_1_Turn
    Button (544,398 29x30), colour toggle: GVL.Turnable_1_Roll_menos, pressed state: GVL.Turnable_1_Roll_menos
        OnMouseClick: toggle GVL.Turnable_1_Roll_menos
    Image (547,402 23x22), "-", colour toggle: GVL.Turnable_1_Roll_menos, image: VisuSymbols.Symbols.ArrowRoundRightLeft
        OnMouseClick: toggle GVL.Turnable_1_Roll_menos
    RoundedRectangle (494,433 29x30), "BL", colour toggle: GVL.Turnable_1_Back_Limit
    Group (527,433 29x30), colour toggle: GVL.Turnable_1_Limit_90
        RoundedRectangle (0,0 29x30), colour toggle: GVL.Diffuse_Sensor_4
        Image (3,4 23x22), image: VisuSymbols.Symbols.DoubleArrow3
    Group (560,433 29x30), colour toggle: GVL.Turnable_1_Limit_0
        RoundedRectangle (0,0 29x30), colour toggle: GVL.Diffuse_Sensor_4
        Image (4,4 23x22), image: VisuSymbols.Symbols.DoubleArrow4
    RoundedRectangle (852,433 29x30), "FL", colour toggle: GVL.Turnable_1_Front_Limit
    RoundedRectangle (885,433 29x30), "BL", colour toggle: GVL.Turnable_1_Back_Limit
    Group (918,433 29x30), colour toggle: GVL.Turnable_1_Limit_90
        RoundedRectangle (0,0 29x30), colour toggle: GVL.Diffuse_Sensor_4
        Image (3,4 23x22), image: VisuSymbols.Symbols.DoubleArrow3
    Group (951,433 29x30), colour toggle: GVL.Turnable_1_Limit_0
        RoundedRectangle (0,0 29x30), colour toggle: GVL.Diffuse_Sensor_4
        Image (4,4 23x22), image: VisuSymbols.Symbols.DoubleArrow4
    Button (869,398 29x30), colour toggle: GVL.Turnable_2_Roll_mas, pressed state: GVL.Turnable_2_Roll_mas
        OnMouseClick: toggle GVL.Turnable_2_Roll_mas
    Image (873,402 23x22), "+", colour toggle: GVL.Turnable_2_Roll_mas, image: VisuSymbols.Symbols.ArrowRoundRightRight
        OnMouseClick: toggle GVL.Turnable_2_Roll_mas
    Button (902,398 29x30), colour toggle: GVL.Turnable_2_Turn, pressed state: GVL.Turnable_2_Turn
        OnMouseClick: toggle GVL.Turnable_2_Turn
    Image (905,402 23x22), colour toggle: GVL.Turnable_2_Turn, image: VisuSymbols.Symbols.ArrowCircle2LeftUpDown
        OnMouseClick: toggle GVL.Turnable_2_Turn
    Button (935,398 29x30), colour toggle: GVL.Turnable_2_Roll_menos, pressed state: GVL.Turnable_2_Roll_menos
        OnMouseClick: toggle GVL.Turnable_2_Roll_menos
    Image (938,402 23x22), "-", colour toggle: GVL.Turnable_2_Roll_menos, image: VisuSymbols.Symbols.ArrowRoundRightLeft
        OnMouseClick: toggle GVL.Turnable_2_Roll_menos
    Line (1023,226) (1070,258)
    Group (1207,130 29x30), colour toggle: GVL.Stacker_Crane_1_Lift
        OnMouseClick: toggle GVL.Stacker_Crane_1_Lift
        Button (0,0 29x30), colour toggle: GVL.Palletizer_1_Open_Plate, pressed state: GVL.Palletizer_1_Open_Plate
        Image (4,3 22x23), image: VisuSymbols.Symbols.ArrowBoldUp
    Group (1240,129 29x30), colour toggle: GVL.Stacker_Crane_1_Right
        OnMouseClick: toggle GVL.Stacker_Crane_1_Right
        Button (0,0 29x30), colour toggle: GVL.Stacker_Crane_1_Right, pressed state: GVL.Palletizer_1_Open_Plate
            OnMouseClick: toggle GVL.Stacker_Crane_1_Right
        Image (4,4 22x23), image: VisuSymbols.Symbols.ArrowBoldRight
    Group (1275,129 29x30), colour toggle: GVL.Stacker_Crane_1_Left
        OnMouseClick: toggle GVL.Stacker_Crane_1_Left
        Button (0,0 29x30), colour toggle: GVL.Palletizer_1_Open_Plate, pressed state: GVL.Palletizer_1_Open_Plate
        Image (3,4 22x23), image: VisuSymbols.Symbols.ArrowBoldLeft
    Group (1207,164 29x30), colour toggle: GVL.Stacker_Crane_1_Moving_Z
        RoundedRectangle (0,0 29x30), colour toggle: GVL.Diffuse_Sensor_4
        Image (4,4 23x22), image: VisuSymbols.Symbols.DoubleArrow4
    Group (1240,164 29x30), colour toggle: GVL.Stacker_Crane_1_Right_Limit
        RoundedRectangle (0,0 29x30), colour toggle: GVL.Diffuse_Sensor_4
        Image (4,4 23x22), image: VisuSymbols.Symbols.ArrowBoldRight
    Group (1173,164 29x30), colour toggle: GVL.Stacker_Crane_1_Moving_X
        RoundedRectangle (0,0 29x30), colour toggle: GVL.Diffuse_Sensor_4
        Image (3,4 23x22), image: VisuSymbols.Symbols.DoubleArrow3
    Group (1309,164 29x30), colour toggle: GVL.Stacker_Crane_1_Middle_Limit
        RoundedRectangle (0,0 29x30), colour toggle: GVL.Diffuse_Sensor_4
        Image (4,3 22x23), image: VisuSymbols.Symbols.Download
    Group (1275,164 29x30), colour toggle: GVL.Stacker_Crane_1_Left_Limit
        RoundedRectangle (0,0 29x30), colour toggle: GVL.Diffuse_Sensor_4
        Image (3,4 22x23), image: VisuSymbols.Symbols.ArrowBoldLeft
    Rectangle (1899,642 178x262), angle 90
    Rectangle (805,107 29x29), "%i", text variable: GVL.RFID_Reader_1_Command_ID
        p4168582468: GVL.RFID_Reader_1_Command_ID
    Rectangle (776,87 82x16), "Command ID"
    Rectangle (778,142 82x16), "Status"
    Rectangle (778,195 82x16), "Read Data"
    Rectangle (805,161 29x29), "%i", text variable: GVL.RFID_Reader_1_Status
        p4168582468: GVL.RFID_Reader_1_Status
    Rectangle (805,217 29x29), "%i", text variable: GVL.RFID_Reader_1_Read_Data
        p4168582468: GVL.RFID_Reader_1_Read_Data
    PowerSwitch (979,155 35x35), variable: GVL.RFID_Reader_1_Ejecute_Comm, behaviour: TOGGLE, style: Switch-PowerSwitch-Gray
    Rectangle (875,87 82x16), "Command"
    Rectangle (875,142 82x16), "Write Data"
    Rectangle (875,195 82x16), "Memory Index"
    Group (901,107 29x30)
        OnMouseClick: write GVL.RFID_Reader_4_Command_ID via VisuDialogs.Numpad, min 0, max 100, format %i
        Button (0,0 29x30), text variable: GVL.RFID_Reader_1_Command
            OnMouseClick: write GVL.RFID_Reader_4_Command_ID via VisuDialogs.Numpad, min 0, max 100, format %i
        Image (5,5 22x22), image: VisuSymbols.Symbols.Edit
    Group (901,161 29x30)
        OnMouseClick: write GVL.RFID_Reader_4_Write_Data via VisuDialogs.Numpad, min 0, max 100, format %i
        Button (0,0 29x30), text variable: GVL.RFID_Reader_1_Command
            OnMouseClick: write GVL.RFID_Reader_4_Command_ID via VisuDialogs.Numpad, min 0, max 100, format %i
        Image (5,5 22x22), image: VisuSymbols.Symbols.Edit
    Group (901,217 29x30)
        OnMouseClick: write GVL.RFID_Reader_4_Memory_Index via VisuDialogs.Numpad, min 0, max 100, format %i
        Button (0,0 29x30), text variable: GVL.RFID_Reader_1_Command
            OnMouseClick: write GVL.RFID_Reader_4_Command_ID via VisuDialogs.Numpad, min 0, max 100, format %i
        Image (5,5 22x22), image: VisuSymbols.Symbols.Edit
    Rectangle (2440,466 153x409), angle 90
    Rectangle (1421,102 248x30), "Almacén"
    Rectangle (2449,456 103x368), angle 90
    PushSwitch (1487,188 50x50), variable: GVL.Emergency_Stop_9, behaviour: TOGGLE, style: Switch-PushSwitch-Red
    Rectangle (1433,159 177x23), "Emergency Stop"
    Lamp1 (1657,190 50x50), variable: NOT GVL.Safety_Door_13 OR NOT GVL.Safety_Door_14 OR NOT GVL.Safety_Door_15, style: Lamp-Lamp1-Yellow
    Rectangle (1625,159 140x23), "Open_Door"
END_VISUALIZATION

// ---- VISUs/Manual/Linea_Produccion_Azul_1.TcVIS
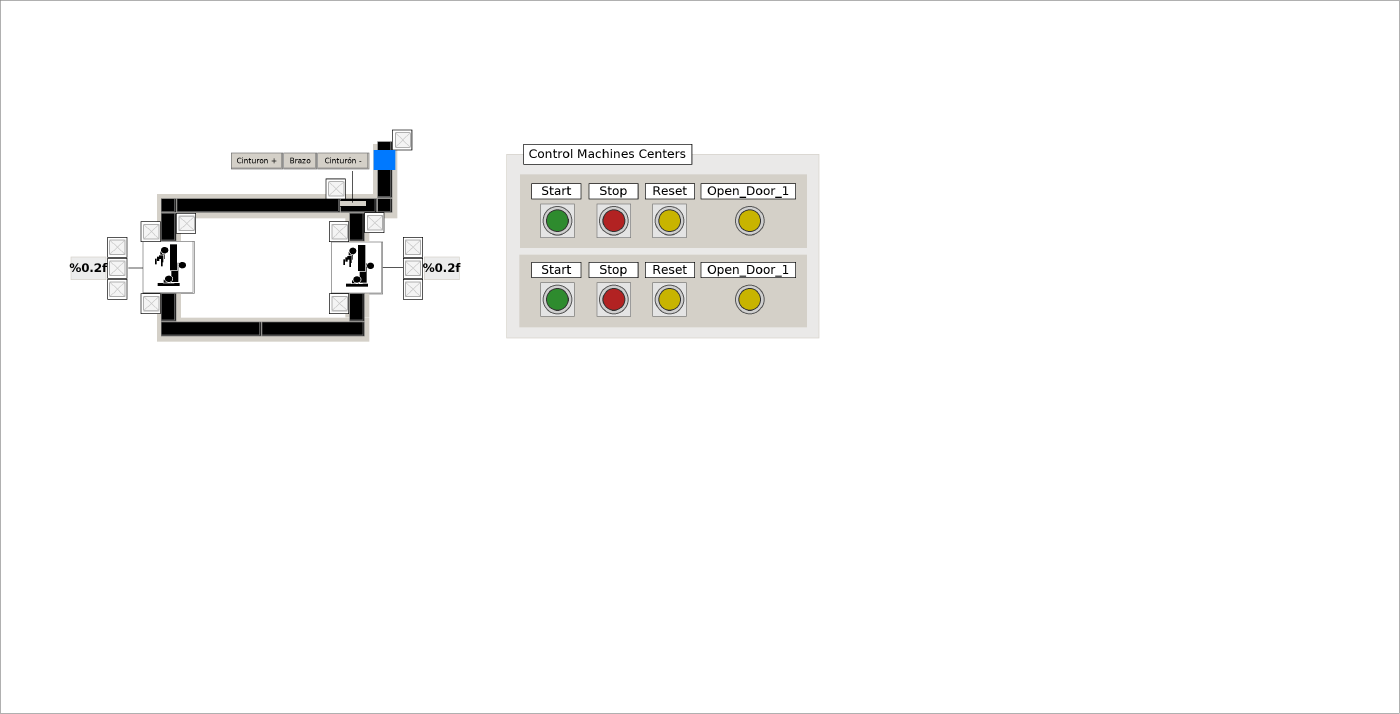
VISUALIZATION Linea_Produccion_Azul_1  // 2060x1052
    Group (487,356 76x81), "2"
        Button (0,0 76x77), pressed state: GVL.Machining_Center_2_Produce_Lids
        RoundedRectangle (35,47 6x34), angle 90
        RoundedRectangle (35,51 6x16), angle 90
        RoundedRectangle (41,31 12x30), angle 47
        Ellipse (32,50 12x11)
        RoundedRectangle (39,4 12x40), angle 130
        Ellipse (52,30 12x11)
        RoundedRectangle (25,11 8x16), angle 24
        Ellipse (26,8 12x11)
        RoundedRectangle (23,20 8x7), angle 24
        RoundedRectangle (27,25 3x6), angle 349
        RoundedRectangle (27,29 2x8), angle 40
        RoundedRectangle (21,23 3x6), angle 259
        RoundedRectangle (18,26 2x8)
    InvisibleInput (82,688 76x76)
    Rectangle (231,286 353x35)
    Rectangle (549,212 35x81)
    Rectangle (231,468 312x35)
    Rectangle (509,321 35x35), angle 90
    Rectangle (230,321 38x35), angle 90
    Group (210,355 76x81), "1"
        Button (0,0 76x77), pressed state: GVL.Machining_Center_1_Produce_Lids
        RoundedRectangle (35,47 6x34), angle 90
        RoundedRectangle (35,51 6x16), angle 90
        RoundedRectangle (41,31 12x30), angle 47
        Ellipse (32,50 12x11)
        RoundedRectangle (39,4 12x40), angle 130
        Ellipse (52,30 12x11)
        RoundedRectangle (25,11 8x16), angle 24
        Ellipse (26,8 12x11)
        RoundedRectangle (23,20 8x7), angle 24
        RoundedRectangle (27,25 3x6), angle 349
        RoundedRectangle (27,29 2x8), angle 40
        RoundedRectangle (21,23 3x6), angle 259
        RoundedRectangle (18,26 2x8)
    Rectangle (509,432 35x35), angle 90
    Rectangle (230,434 38x35), angle 90
    Line (563,394) (593,394)
    Line (210,395) (189,395)
    Rectangle (1789,525 271x460), angle 90
    Rectangle (770,212 248x30), "Control Machines Centers"
    Rectangle (1798,512 108x422), angle 90
    PushSwitch (795,300 50x50), variable: GVL.Machining_Center_1_Start, behaviour: TOGGLE, style: Switch-PushSwitch-Green
    Rectangle (782,270 73x23), "Start"
    Lamp1 (1078,300 50x50), variable: GVL.Diffuse_Sensor_45, style: Lamp-Lamp1-Yellow
    Rectangle (1031,270 140x23), "Open_Door_1"
    Rectangle (1797,629 107x423), angle 90
    InvisibleInput (1018,652 49x69)
    InvisibleInput (1267,179 49x69)
    InvisibleInput (1090,651 49x69)
    InvisibleInput (1264,0 49x69)
    InvisibleInput (1265,68 49x69)
    Button (555,208 22x83), colour toggle: GVL.Belt_Conveyor_2m_3, pressed state: GVL.Belt_Conveyor_2m_3
        OnMouseClick: toggle GVL.Belt_Conveyor_2m_3
    Group (577,191 29x30), colour toggle: GVL.Diffuse_Sensor_5
        RoundedRectangle (0,0 29x30), colour toggle: GVL.Diffuse_Sensor_4
        Image (4,4 23x22), image: VisuSymbols.Symbols.RSS1
    RoundedRectangle (550,221 31x29)
    Button (555,292 22x21), colour toggle: GVL.Curved_Belt_Conveyor_1_CW, pressed state: GVL.Curved_Belt_Conveyor_1_CW
        OnMouseClick: toggle GVL.Curved_Belt_Conveyor_1_CW
    Button (501,292 53x21), colour toggle: GVL.Belt_Conveyor_2m_4, pressed state: GVL.Belt_Conveyor_2m_4
        OnMouseClick: toggle GVL.Belt_Conveyor_2m_4
    Rectangle (499,295 40x9), angle -45
    Button (260,292 240x21), colour toggle: GVL.Belt_Conveyor_6m_2, pressed state: GVL.Belt_Conveyor_6m_2
        OnMouseClick: toggle GVL.Belt_Conveyor_6m_2
    Button (237,292 22x21), colour toggle: GVL.Curved_Belt_Conveyor_1_CCW, pressed state: GVL.Curved_Belt_Conveyor_1_CCW
        OnMouseClick: toggle GVL.Curved_Belt_Conveyor_1_CCW
    Button (237,314 22x41), colour toggle: GVL.Belt_Conveyor_2m_6, pressed state: GVL.Belt_Conveyor_2m_6
        OnMouseClick: toggle GVL.Belt_Conveyor_2m_6
    Button (514,314 22x41), colour toggle: GVL.Belt_Conveyor_2m_5, pressed state: GVL.Belt_Conveyor_2m_5
        OnMouseClick: toggle GVL.Belt_Conveyor_2m_5
    Button (514,432 22x41), colour toggle: GVL.Belt_Conveyor_2m_14, pressed state: GVL.Belt_Conveyor_2m_14
        OnMouseClick: toggle GVL.Belt_Conveyor_2m_14
    Button (237,432 22x41), colour toggle: GVL.Belt_Conveyor_2m_13, pressed state: GVL.Belt_Conveyor_2m_13
        OnMouseClick: toggle GVL.Belt_Conveyor_2m_13
    Button (237,474 147x21), colour toggle: GVL.Belt_Conveyor_4m_4, pressed state: GVL.Belt_Conveyor_4m_4
        OnMouseClick: toggle GVL.Belt_Conveyor_4m_4
    Button (385,474 151x21), colour toggle: GVL.Belt_Conveyor_4m_5, pressed state: GVL.Belt_Conveyor_4m_5
        OnMouseClick: toggle GVL.Belt_Conveyor_4m_5
    Button (417,225 49x24), "Brazo", colour toggle: GVL.Pivot_Arm_Sorter_2_Turn, pressed state: GVL.Pivot_Arm_Sorter_2_Turn
        OnMouseClick: toggle GVL.Pivot_Arm_Sorter_2_Turn
    Button (340,225 76x24), "Cinturon +", colour toggle: GVL.Pivot_Arm_Sorter_2_Belt_mas, pressed state: GVL.Pivot_Arm_Sorter_2_Belt_mas
        OnMouseClick: toggle GVL.Pivot_Arm_Sorter_2_Belt_mas
    Button (467,225 76x24), "Cinturón -", colour toggle: GVL.Pivot_Arm_Sorter_2_Belt_menos, pressed state: GVL.Pivot_Arm_Sorter_2_Belt_menos
        OnMouseClick: toggle GVL.Pivot_Arm_Sorter_2_Belt_menos
    Line (518,252) (518,298)
    Group (479,263 29x30), colour toggle: GVL.Diffuse_Sensor_6
        RoundedRectangle (0,0 29x30), colour toggle: GVL.Diffuse_Sensor_4
        Image (4,4 23x22), image: VisuSymbols.Symbols.RSS1
    Group (536,313 29x30), colour toggle: GVL.Diffuse_Sensor_7
        RoundedRectangle (0,0 29x30), colour toggle: GVL.Diffuse_Sensor_4
        Image (4,4 23x22), image: VisuSymbols.Symbols.RSS1
    Group (259,314 29x30), colour toggle: GVL.Diffuse_Sensor_8
        RoundedRectangle (0,0 29x30), colour toggle: GVL.Diffuse_Sensor_4
        Image (4,4 23x22), image: VisuSymbols.Symbols.RSS1
    Group (207,432 29x30), colour toggle: GVL.Diffuse_Sensor_17
        RoundedRectangle (0,0 29x30), colour toggle: GVL.Diffuse_Sensor_4
        Image (4,4 23x22), image: VisuSymbols.Symbols.RSS1
    Group (484,432 29x30), colour toggle: GVL.Diffuse_Sensor_18
        RoundedRectangle (0,0 29x30), colour toggle: GVL.Diffuse_Sensor_4
        Image (4,4 23x22), image: VisuSymbols.Symbols.RSS1
    Group (207,326 29x30), colour toggle: GVL.Diffuse_Sensor_15
        RoundedRectangle (0,0 29x30), colour toggle: GVL.Diffuse_Sensor_4
        Image (4,4 23x22), image: VisuSymbols.Symbols.RSS1
    Group (484,326 29x30), colour toggle: GVL.Diffuse_Sensor_16
        RoundedRectangle (0,0 29x30), colour toggle: GVL.Diffuse_Sensor_4
        Image (4,4 23x22), image: VisuSymbols.Symbols.RSS1
    Rectangle (104,378 52x34), "%0.2f", text variable: GVL.Machining_Center_1_Progress
        p4168582468: GVL.Machining_Center_1_Progress
    Group (158,380 29x30), colour toggle: GVL.Machining_Center_1_IsBusy
        RoundedRectangle (0,0 29x30), colour toggle: GVL.Diffuse_Sensor_4
        Image (3,4 23x22), image: VisuSymbols.Symbols.Wheel
    Group (158,349 29x30), colour toggle: GVL.Machining_Center_1_Error
        RoundedRectangle (0,0 29x30), colour toggle: GVL.Diffuse_Sensor_4
        Image (3,4 23x22), image: VisuSymbols.Symbols.Bell
    Group (158,411 29x30), colour toggle: GVL.Machining_Center_1_Opened
        RoundedRectangle (0,0 29x30), colour toggle: GVL.Diffuse_Sensor_4
        Image (3,4 23x22), image: VisuSymbols.Symbols.DoubleArrow3
    Rectangle (624,378 52x34), "%0.2f", text variable: GVL.Machining_Center_1_Progress
        p4168582468: GVL.Machining_Center_1_Progress
    Group (593,380 29x30), colour toggle: GVL.Machining_Center_2_IsBusy
        RoundedRectangle (0,0 29x30), colour toggle: GVL.Diffuse_Sensor_4
        Image (3,4 23x22), image: VisuSymbols.Symbols.Wheel
    Group (593,349 29x30), colour toggle: GVL.Machining_Center_2_Error
        RoundedRectangle (0,0 29x30), colour toggle: GVL.Diffuse_Sensor_4
        Image (3,4 23x22), image: VisuSymbols.Symbols.Bell
    Group (593,411 29x30), colour toggle: GVL.Machining_Center_2_Opened
        RoundedRectangle (0,0 29x30), colour toggle: GVL.Diffuse_Sensor_4
        Image (3,4 23x22), image: VisuSymbols.Symbols.DoubleArrow3
    Rectangle (866,270 73x23), "Stop"
    Rectangle (949,270 73x23), "Reset"
    PushSwitch (878,300 50x50), variable: GVL.Machine_Center_1_Stop, behaviour: TOGGLE, style: Switch-PushSwitch-Red
    PushSwitch (960,300 50x50), variable: GVL.Machine_Center_1_Reset, behaviour: TOGGLE, style: Switch-PushSwitch-Yellow
    PushSwitch (795,416 50x50), variable: GVL.Machining_Center_2_Start, behaviour: TOGGLE, style: Switch-PushSwitch-Green
    Rectangle (782,386 73x23), "Start"
    Lamp1 (1078,416 50x50), variable: GVL.Diffuse_Sensor_46, style: Lamp-Lamp1-Yellow
    Rectangle (1031,386 140x23), "Open_Door_1"
    Rectangle (866,386 73x23), "Stop"
    Rectangle (949,386 73x23), "Reset"
    PushSwitch (878,416 50x50), variable: GVL.Machine_Center_2_Stop, behaviour: TOGGLE, style: Switch-PushSwitch-Red
    PushSwitch (960,416 50x50), variable: GVL.Machine_Center_2_Reset, behaviour: TOGGLE, style: Switch-PushSwitch-Yellow
END_VISUALIZATION

// ---- VISUs/Manual/Linea_Produccion_Azul_2.TcVIS
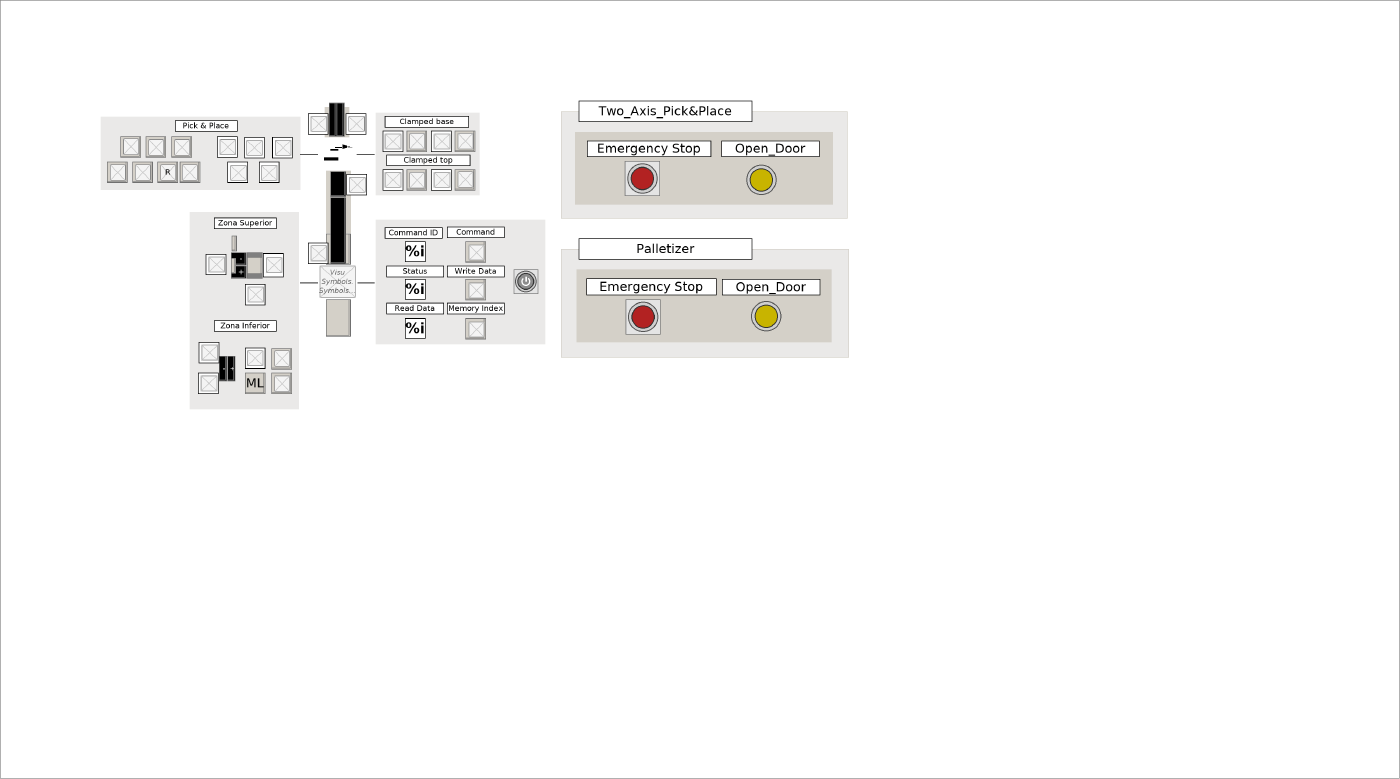
VISUALIZATION Linea_Produccion_Azul_2  // 2001x1114
    Rectangle (1846,508 153x409), angle 90
    Rectangle (827,144 248x30), "Two_Axis_Pick&Place"
    Rectangle (1855,498 103x368), angle 90
    PushSwitch (893,230 50x50), variable: GVL.Emergency_Stop_3, behaviour: TOGGLE, style: Switch-PushSwitch-Red
    Rectangle (839,201 177x23), "Emergency Stop"
    Lamp1 (1063,232 50x50), variable: NOT GVL.Safety_Door_1 OR NOT GVL.Safety_Door_2, style: Lamp-Lamp1-Yellow
    Rectangle (1031,201 140x23), "Open_Door"
    Rectangle (1846,703 155x411), angle 90
    Rectangle (827,341 248x30), "Palletizer"
    Rectangle (1614,447 104x364), angle 90
    PushSwitch (894,428 50x50), behaviour: TOGGLE, style: Switch-PushSwitch-Red
    Rectangle (838,398 186x24), "Emergency Stop"
    Lamp1 (1070,427 50x50), variable: NOT GVL.Safety_Door_3 OR NOT GVL.Safety_Door_4, style: Lamp-Lamp1-Yellow
    Rectangle (1032,399 140x23), "Open_Door"
    InvisibleInput (880,700 18x108)
    InvisibleInput (1316,220 49x41)
    Rectangle (1327,891 282x156), angle 90
    Rectangle (1569,733 118x148), angle 90
    Rectangle (1340,766 104x285), angle 90
    Button (466,334 35x44), colour toggle: GVL.Roller_Conveyor_2m_1, pressed state: GVL.Roller_Conveyor_2m_1
        OnMouseClick: toggle GVL.Roller_Conveyor_2m_1
    Rectangle (461,157 43x35), angle 90
    Group (456,196 53x49)
        InvisibleInput (0,0 53x49)
        RoundedRectangle (7,29 20x4), angle 107
        RoundedRectangle (16,17 11x2), angle 107
        RoundedRectangle (23,14 11x1), angle 180
        Polygon (33,10) (40,12) (40,14) (40,15) (33,17)
        Polygon (47,14) (47,14) (41,14) (41,14) (41,13)
    Rectangle (440,271 89x35), angle 90
    Group (455,378 55x50)
        InvisibleInput (0,0 55x50)
        Image (2,2 51x45), image: VisuSymbols.Symbols.Box
    Line (429,220) (454,220)
    Line (429,404) (454,404)
    Line (511,404) (535,404)
    Button (470,147 11x48), colour toggle: GVL.Belt_Conveyor_4m_6, pressed state: GVL.Belt_Conveyor_4m_6
        OnMouseClick: toggle GVL.Belt_Conveyor_4m_6
    Button (481,147 11x48), colour toggle: GVL.Belt_Conveyor_4m_7, pressed state: GVL.Belt_Conveyor_4m_7
        OnMouseClick: toggle GVL.Belt_Conveyor_4m_7
    Button (472,245 22x36), colour toggle: GVL.Belt_Conveyor_2m_15, pressed state: GVL.Belt_Conveyor_2m_15
        OnMouseClick: toggle GVL.Belt_Conveyor_2m_15
    Button (472,282 22x95), colour toggle: GVL.Belt_Conveyor_Inclined_1, pressed state: GVL.Belt_Conveyor_Inclined_1
        OnMouseClick: toggle GVL.Belt_Conveyor_Inclined_1
    Button (466,428 35x53), colour toggle: GVL.Roller_Conveyor_2m_2, pressed state: GVL.Roller_Conveyor_2m_2
        OnMouseClick: toggle GVL.Roller_Conveyor_2m_2
    Group (440,162 29x30), colour toggle: GVL.Diffuse_Sensor_12
        RoundedRectangle (0,0 29x30), colour toggle: GVL.Diffuse_Sensor_4
        Image (4,4 23x22), image: VisuSymbols.Symbols.RSS1
    Group (494,162 29x30), colour toggle: GVL.Diffuse_Sensor_13
        RoundedRectangle (0,0 29x30), colour toggle: GVL.Diffuse_Sensor_4
        Image (4,4 23x22), image: VisuSymbols.Symbols.RSS1
    Group (495,249 29x30), colour toggle: GVL.Diffuse_Sensor_14
        RoundedRectangle (0,0 29x30), colour toggle: GVL.Diffuse_Sensor_4
        Image (4,4 23x22), image: VisuSymbols.Symbols.RSS1
    Group (440,347 29x30), colour toggle: GVL.Diffuse_Sensor_22
        RoundedRectangle (0,0 29x30), colour toggle: GVL.Diffuse_Sensor_4
        Image (4,4 23x22), image: VisuSymbols.Symbols.RSS1
    Group (310,195 29x30), colour toggle: GVL.Two_Axis_Pick_Place_1_Detected
        RoundedRectangle (0,0 29x30), colour toggle: GVL.Two_Axis_Pick_Place_1_Detected
        Image (4,4 23x22), image: VisuSymbols.Symbols.RSS1
    Group (349,196 29x30), colour toggle: GVL.Two_Axis_Pick_Place_1_MovingX
        RoundedRectangle (0,0 29x30), colour toggle: GVL.Diffuse_Sensor_4
        Image (3,4 23x22), image: VisuSymbols.Symbols.DoubleArrow3
    Group (325,231 29x30), "G", colour toggle: GVL.Two_Axis_Pick_Place_1_Gripper_Rotating
        RoundedRectangle (0,0 29x30), colour toggle: GVL.Diffuse_Sensor_4
        Image (4,5 23x22), image: VisuSymbols.Symbols.ArrowRoundRightDown
    Group (389,196 29x30), colour toggle: GVL.Two_Axis_Pick_Place_1_MovingZ
        RoundedRectangle (0,0 29x30), colour toggle: GVL.Diffuse_Sensor_4
        Image (4,4 23x22), image: VisuSymbols.Symbols.DoubleArrow4
    Group (370,231 29x30), "R", colour toggle: GVL.Two_Axis_Pick_Place_1_Rotating
        RoundedRectangle (0,0 29x30), colour toggle: GVL.Diffuse_Sensor_4
        Image (3,5 23x22), image: VisuSymbols.Symbols.ArrowHalfLeftUp
    Rectangle (250,172 89x16), "Pick & Place"
    Group (547,187 29x30), colour toggle: NOT GVL.Right_Positioner_1_Clamped
        RoundedRectangle (0,0 29x30), colour toggle: GVL.Diffuse_Sensor_4
        Image (3,4 23x22), image: VisuSymbols.Symbols.DoubleArrow3
    Group (616,187 29x30), colour toggle: GVL.Right_Positioner_1_Limit
        RoundedRectangle (0,0 29x30), colour toggle: GVL.Diffuse_Sensor_4
        Image (4,4 23x22), image: VisuSymbols.Symbols.DoubleArrow4
    Rectangle (550,166 120x16), "Clamped base"
    Group (547,242 29x30), colour toggle: NOT GVL.Right_Positioner_2_Clamped
        RoundedRectangle (0,0 29x30), colour toggle: GVL.Diffuse_Sensor_4
        Image (3,4 23x22), image: VisuSymbols.Symbols.DoubleArrow3
    Group (616,242 29x30), colour toggle: GVL.Right_Positioner_2_Limit
        RoundedRectangle (0,0 29x30), colour toggle: GVL.Diffuse_Sensor_4
        Image (4,4 23x22), image: VisuSymbols.Symbols.DoubleArrow4
    Rectangle (552,221 120x16), "Clamped top"
    Line (510,220) (535,220)
    Button (330,361 22x18), "-", colour toggle: GVL.Palletizer_1_Belt_menos, pressed state: GVL.Palletizer_1_Belt_menos
        OnMouseClick: toggle GVL.Palletizer_1_Belt_menos
    Button (331,337 7x22), colour toggle: GVL.Palletizer_1_Turn, pressed state: GVL.Palletizer_1_Turn
        OnMouseClick: toggle GVL.Palletizer_1_Turn
    Button (353,361 22x36), colour toggle: GVL.Palletizer_1_Open_Plate, pressed state: GVL.Palletizer_1_Open_Plate
        OnMouseClick: toggle GVL.Palletizer_1_Open_Plate
    Button (353,391 22x7), colour toggle: GVL.Palletizer_1_Clamb, pressed state: GVL.Palletizer_1_Clamb
        OnMouseClick: toggle GVL.Palletizer_1_Clamb
    Group (350,406 29x30), colour toggle: GVL.Palletizer_1_Clamped
        RoundedRectangle (0,0 29x30), colour toggle: GVL.Diffuse_Sensor_4
        Image (4,4 23x22), image: VisuSymbols.Symbols.DoubleArrow4
    Group (376,362 29x34), colour toggle: GVL.Palletizer_1_Plate_Limit
        RoundedRectangle (0,0 29x34), colour toggle: GVL.Diffuse_Sensor_4
        Image (4,6 23x22), angle 45, image: VisuSymbols.Symbols.DoubleArrow1
    Button (330,380 22x18), "+", colour toggle: GVL.Palletizer_1_Belt_mas, pressed state: GVL.Palletizer_1_Belt_mas
        OnMouseClick: toggle GVL.Palletizer_1_Belt_mas
    Button (330,369 7x22), colour toggle: GVL.Palletizer_1_Push, pressed state: GVL.Palletizer_1_Push
        OnMouseClick: toggle GVL.Palletizer_1_Push
    Button (353,361 22x7), colour toggle: GVL.Palletizer_1_Clamb, pressed state: GVL.Palletizer_1_Clamb
        OnMouseClick: toggle GVL.Palletizer_1_Clamb
    Group (294,363 29x30), colour toggle: GVL.Palletizer_1_Pusher_Limit
        RoundedRectangle (0,0 29x30), colour toggle: GVL.Diffuse_Sensor_4
        Image (4,4 23x22), image: VisuSymbols.Symbols.ArrowBoldRight
    Button (325,509 11x36), "+", colour toggle: GVL.Palletizer_1_Chain_mas, pressed state: GVL.Palletizer_1_Belt_mas
        OnMouseClick: toggle GVL.Palletizer_1_Chain_mas
    Button (313,509 11x36), "-", colour toggle: GVL.Palletizer_1_Chain_menos, pressed state: GVL.Palletizer_1_Belt_menos
        OnMouseClick: toggle GVL.Palletizer_1_Chain_menos
    Group (284,489 29x30), colour toggle: GVL.Palletizer_1_Elevator_Back_Limit
        RoundedRectangle (0,0 29x30), colour toggle: GVL.Two_Axis_Pick_Place_1_Detected
        Image (4,4 23x22), image: VisuSymbols.Symbols.RSS1
    Group (283,533 29x30), colour toggle: GVL.Palletizer_1_Elevator_Front_Limit
        RoundedRectangle (0,0 29x30), colour toggle: GVL.Two_Axis_Pick_Place_1_Detected
        Image (4,4 23x22), image: VisuSymbols.Symbols.RSS1
    Group (350,497 29x30), colour toggle: GVL.Palletizer_1_Elevator_Moving
        RoundedRectangle (0,0 29x30), colour toggle: GVL.Diffuse_Sensor_4
        Image (3,4 23x22), image: VisuSymbols.Symbols.Wheel
    Button (350,533 29x30), "ML", colour toggle: GVL.Palletizer_1_Elevator_Move_Limit, pressed state: GVL.Palletizer_1_Open_Plate
        OnMouseClick: toggle GVL.Palletizer_1_Elevator_Move_Limit
    Group (388,498 29x30), colour toggle: GVL.Palletizer_1_Elevator_mas
        OnMouseClick: toggle GVL.Palletizer_1_Elevator_mas
        Button (0,0 29x30)
        Image (4,3 22x23), image: VisuSymbols.Symbols.ArrowBoldUp
    Group (388,533 29x30), colour toggle: GVL.Palletizer_1_Elevator_menos
        OnMouseClick: toggle GVL.Palletizer_1_Elevator_menos
        Button (0,0 29x30)
        Image (4,4 22x23), image: VisuSymbols.Symbols.ArrowBoldDown
    Rectangle (306,311 89x16), "Zona Superior"
    Rectangle (306,458 89x16), "Zona Inferior"
    Group (208,195 29x30), colour toggle: GVL.Two_Axis_Pick_Place_1X
        OnMouseClick: toggle GVL.Two_Axis_Pick_Place_1X
        Button (0,0 29x30)
        Image (4,4 22x23), image: VisuSymbols.Symbols.ArrowBoldRight
    Group (172,195 29x30), colour toggle: GVL.Two_Axis_Pick_Place_1_Grab
        OnMouseClick: toggle GVL.Two_Axis_Pick_Place_1_Grab
        Button (0,0 29x30)
        Image (4,3 22x23), image: VisuSymbols.Symbols.Download
    Group (257,231 29x30), colour toggle: GVL.Two_Axis_Pick_Place_1_Rotate_CCW
        OnMouseClick: toggle GVL.Two_Axis_Pick_Place_1_Rotate_CCW
        Button (0,0 29x30)
        Image (3,4 22x23), image: VisuSymbols.Symbols.ArrowHalfLeftUp
    Group (189,231 29x30), colour toggle: GVL.Two_Axis_Pick_Place_1_Gripper_CW
        OnMouseClick: toggle GVL.Two_Axis_Pick_Place_1_Gripper_CW
        Button (0,0 29x30)
        Image (4,4 22x23), image: VisuSymbols.Symbols.ArrowRoundRightDown
    Group (153,231 29x30), colour toggle: GVL.Two_Axis_Pick_Place_1_Gripper_CCW
        OnMouseClick: toggle GVL.Two_Axis_Pick_Place_1_Gripper_CCW
        Button (0,0 29x30)
        Image (4,4 22x23), image: VisuSymbols.Symbols.ArrowRoundLeftBottom
    Group (225,231 29x30), colour toggle: GVL.Two_Axis_Pick_Place_1_Rotare_CW
        OnMouseClick: toggle GVL.Two_Axis_Pick_Place_1_Rotare_CW
        Button (0,0 29x30)
        Image (4,4 22x23), "R", colour toggle: GVL.Two_Axis_Pick_Place_1_Rotate_CW, image: VisuSymbols.Symbols.ArrowHalfRightUp
            OnMouseClick: toggle GVL.Two_Axis_Pick_Place_1_Rotate_CW
    Group (245,195 29x30), colour toggle: GVL.Two_Axis_Pick_Place_1Z
        OnMouseClick: toggle GVL.Two_Axis_Pick_Place_1Z
        Button (0,0 29x30)
        Image (4,4 22x23), image: VisuSymbols.Symbols.ArrowBoldDown
    Group (581,187 29x30), colour toggle: GVL.Right_Positioner_1_Clamp
        OnMouseClick: toggle GVL.Right_Positioner_1_Clamp
        Button (0,0 29x30)
        Image (4,3 22x23), image: VisuSymbols.Symbols.DoubleArrow3
    Group (581,242 29x30), colour toggle: GVL.Right_Positioner_2_Clamp
        OnMouseClick: toggle GVL.Right_Positioner_2_Clamp
        Button (0,0 29x30)
        Image (4,4 22x23), image: VisuSymbols.Symbols.DoubleArrow3
    Group (650,242 29x30), colour toggle: GVL.Right_Positioner_2_Raise
        OnMouseClick: toggle GVL.Right_Positioner_2_Raise
        Button (0,0 29x30)
        Image (4,3 22x23), image: VisuSymbols.Symbols.ArrowBoldUp
    Group (650,187 29x30), colour toggle: GVL.Right_Positioner_1_Raise
        OnMouseClick: toggle GVL.Right_Positioner_1_Raise
        Button (0,0 29x30)
        Image (4,3 22x23), image: VisuSymbols.Symbols.ArrowBoldUp
    Rectangle (1569,792 178x242), angle 90
    Rectangle (579,345 29x29), "%i", text variable: GVL.RFID_Reader_1_Command_ID
        p4168582468: GVL.RFID_Reader_1_Command_ID
    Rectangle (550,325 82x16), "Command ID"
    Rectangle (552,380 82x16), "Status"
    Rectangle (552,433 82x16), "Read Data"
    Rectangle (579,399 29x29), "%i", text variable: GVL.RFID_Reader_1_Status
        p4168582468: GVL.RFID_Reader_1_Status
    Rectangle (579,455 29x29), "%i", text variable: GVL.RFID_Reader_1_Read_Data
        p4168582468: GVL.RFID_Reader_1_Read_Data
    PowerSwitch (734,385 35x35), variable: GVL.RFID_Reader_1_Ejecute_Comm, behaviour: TOGGLE, style: Switch-PowerSwitch-Gray
    Rectangle (639,324 82x16), "Command"
    Rectangle (639,380 82x16), "Write Data"
    Rectangle (639,433 82x16), "Memory Index"
    Group (665,345 29x30)
        OnMouseClick: write GVL.RFID_Reader_1_Command_ID via VisuDialogs.Numpad, min 0, max 100, format %i
        Button (0,0 29x30), text variable: GVL.RFID_Reader_1_Command
            OnMouseClick: write GVL.RFID_Reader_4_Command_ID via VisuDialogs.Numpad, min 0, max 100, format %i
        Image (5,5 22x22), image: VisuSymbols.Symbols.Edit
    Group (665,399 29x30)
        OnMouseClick: write GVL.RFID_Reader_1_Write_Data via VisuDialogs.Numpad, min 0, max 100, format %i
        Button (0,0 29x30), text variable: GVL.RFID_Reader_1_Command
            OnMouseClick: write GVL.RFID_Reader_4_Command_ID via VisuDialogs.Numpad, min 0, max 100, format %i
        Image (5,5 22x22), image: VisuSymbols.Symbols.Edit
    Group (665,455 29x30)
        OnMouseClick: write GVL.RFID_Reader_1_Memory_Index via VisuDialogs.Numpad, min 0, max 100, format %i
        Button (0,0 29x30), text variable: GVL.RFID_Reader_1_Command
            OnMouseClick: write GVL.RFID_Reader_4_Command_ID via VisuDialogs.Numpad, min 0, max 100, format %i
        Image (5,5 22x22), image: VisuSymbols.Symbols.Edit
END_VISUALIZATION

// ---- VISUs/HMI.TcVIS
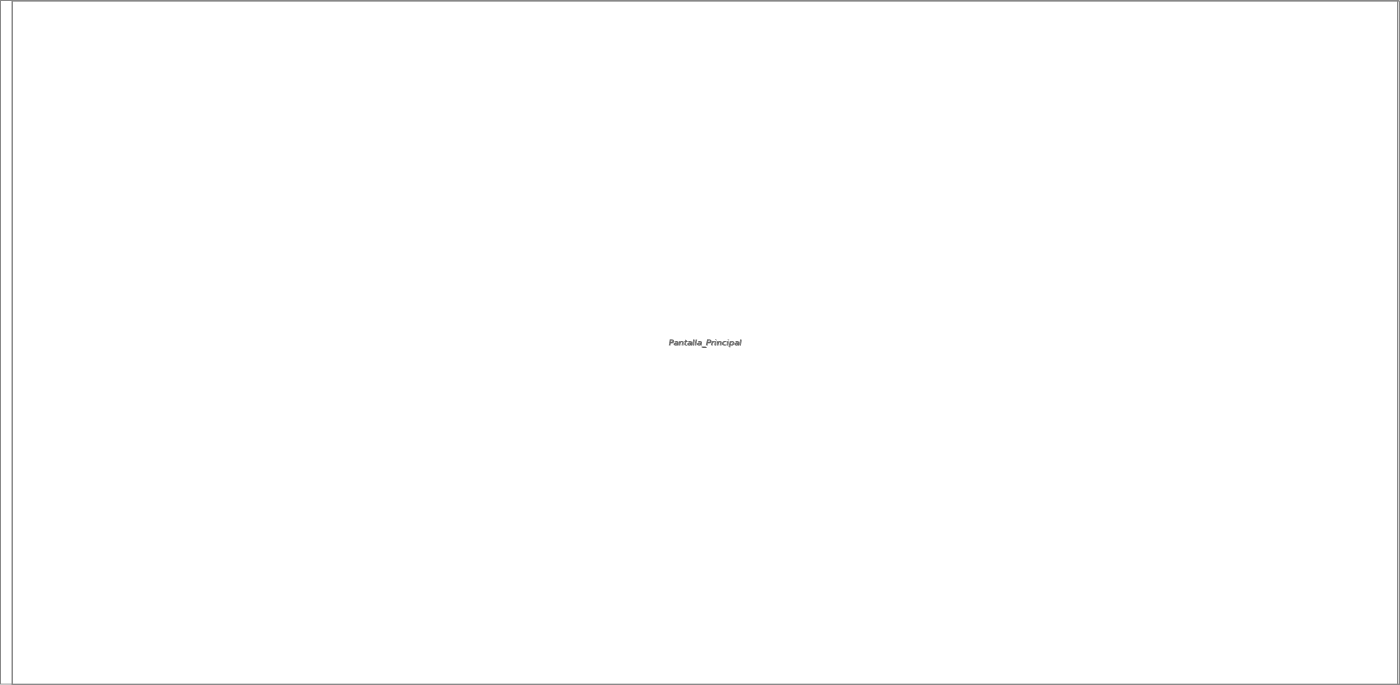
VISUALIZATION HMI  // 1709x837
    TabControl (15,0 1691x837), invisible if: NOT GVL.Manual
        shows Pantalla_Principal()
        shows Entrada_Manual()
        shows Linea_Produccion_Azul_1()
        shows Linea_Produccion_Azul_2()
        shows Linea_Almacen_Manual()
        shows Almacen_Manual()
        shows Senales()
        [0]: TabTitle=Global
        [1]: TabTitle=Entrada
        [2]: TabTitle=Comienzo Producción Azul
        [3]: TabTitle=Final Producción Azul
        [4]: TabTitle=Línea Almacén
        [5]: TabTitle=Entrada Almacen
        [6]: TabTitle=Señales
    TabControl (14,1 1695x836), invisible if: GVL.Manual
        shows Pantalla_Principal()
        shows Entrada_Manual()
        shows Linea_Produccion_Azul_1()
        shows Linea_Produccion_Azul_2()
        shows Linea_Almacen_Manual()
        shows Almacen_Manual()
        shows Senales()
        [0]: TabTitle=Global
        [1]: TabTitle=Entrada
        [2]: TabTitle=Comienzo Linea Azul
        [3]: TabTitle=Final Linea Azul
        [4]: TabTitle=Linea Almacen
        [5]: TabTitle=Entrada Almacen
        [6]: TabTitle=Señales
END_VISUALIZATION
